  LIN {X 2625.059,Y -2566.499,Z 65.775,A 88.24449,B 0.00000,C 180.00000} ; preinsert
  LIN {X 2625.059,Y -2566.499,Z -184.225,A 88.24449,B 0.00000,C 180.00000} ; insert
  LIN {X 2625.059,Y -2566.499,Z -184.225,A 88.24449,B 0.00000,C 180.00000} ; release
  LIN {X 2625.059,Y -2566.499,Z 115.775,A 88.24449,B 0.00000,C 180.00000} ; retreat
  ; Step 1793, bar 2402
  LIN {X 1875.059,Y -2566.499,Z 1020.471,A 88.24449,B 0.00000,C 180.00000} ; outside
  LIN {X 1875.059,Y -2566.499,Z 65.775,A 88.24449,B 0.00000,C 180.00000} ; preinsert
  LIN {X 1875.059,Y -2566.499,Z -184.225,A 88.24449,B 0.00000,C 180.00000} ; insert
  LIN {X 1875.059,Y -2566.499,Z -184.225,A 88.24449,B 0.00000,C 180.00000} ; release
  LIN {X 1875.059,Y -2566.499,Z 115.775,A 88.24449,B 0.00000,C 180.00000} ; retreat
  ; Step 1794, bar 2396
  LIN {X 1125.059,Y -2566.499,Z 1020.471,A 88.24449,B 0.00000,C 180.00000} ; outside
  LIN {X 1125.059,Y -2566.499,Z 65.775,A 88.24449,B 0.00000,C 180.00000} ; preinsert
  LIN {X 1125.059,Y -2566.499,Z -184.225,A 88.24449,B 0.00000,C 180.00000} ; insert
  LIN {X 1125.059,Y -2566.499,Z -184.225,A 88.24449,B 0.00000,C 180.00000} ; release
  LIN {X 1125.059,Y -2566.499,Z 115.775,A 88.24449,B 0.00000,C 180.00000} ; retreat
  ; Step 1795, bar 2391
  LIN {X 375.059,Y -2566.499,Z 1020.471,A 88.24449,B 0.00000,C 180.00000} ; outside
  LIN {X 375.059,Y -2566.499,Z 65.775,A 88.24449,B 0.00000,C 180.00000} ; preinsert
  LIN {X 375.059,Y -2566.499,Z -184.225,A 88.24449,B 0.00000,C 180.00000} ; insert
  LIN {X 375.059,Y -2566.499,Z -184.225,A 88.24449,B 0.00000,C 180.00000} ; release
  LIN {X 375.059,Y -2566.499,Z 115.775,A 88.24449,B 0.00000,C 180.00000} ; retreat
  ; Step 1796, bar 2106
  LIN {X -15850.059,Y 2566.499,Z 1020.471,A -91.75551,B 0.00000,C -180.00000} ; outside
  LIN {X -15850.059,Y 2566.499,Z 65.775,A -91.75551,B 0.00000,C -180.00000} ; preinsert
  LIN {X -15850.059,Y 2566.499,Z -184.225,A -91.75551,B 0.00000,C -180.00000} ; insert
  LIN {X -15850.059,Y 2566.499,Z -184.225,A -91.75551,B 0.00000,C -180.00000} ; release
  LIN {X -15850.059,Y 2566.499,Z 115.775,A -91.75551,B 0.00000,C -180.00000} ; retreat
  ; Step 1797, bar 2100
  LIN {X -15250.059,Y 2566.499,Z 1020.471,A -91.75551,B 0.00000,C -180.00000} ; outside
  LIN {X -15250.059,Y 2566.499,Z 65.775,A -91.75551,B 0.00000,C -180.00000} ; preinsert
  LIN {X -15250.059,Y 2566.499,Z -184.225,A -91.75551,B 0.00000,C -180.00000} ; insert
  LIN {X -15250.059,Y 2566.499,Z -184.225,A -91.75551,B 0.00000,C -180.00000} ; release
  LIN {X -15250.059,Y 2566.499,Z 115.775,A -91.75551,B 0.00000,C -180.00000} ; retreat
  ; Step 1798, bar 2094
  LIN {X -14650.059,Y 2566.499,Z 1020.471,A -91.75551,B 0.00000,C -180.00000} ; outside
  LIN {X -14650.059,Y 2566.499,Z 65.775,A -91.75551,B 0.00000,C -180.00000} ; preinsert
  LIN {X -14650.059,Y 2566.499,Z -184.225,A -91.75551,B 0.00000,C -180.00000} ; insert
  LIN {X -14650.059,Y 2566.499,Z -184.225,A -91.75551,B 0.00000,C -180.00000} ; release
  LIN {X -14650.059,Y 2566.499,Z 115.775,A -91.75551,B 0.00000,C -180.00000} ; retreat
  ; Step 1799, bar 2088
  LIN {X -14050.059,Y 2566.499,Z 1020.471,A -91.75551,B 0.00000,C -180.00000} ; outside
  LIN {X -14050.059,Y 2566.499,Z 65.775,A -91.75551,B 0.00000,C -180.00000} ; preinsert
  LIN {X -14050.059,Y 2566.499,Z -184.225,A -91.75551,B 0.00000,C -180.00000} ; insert
  LIN {X -14050.059,Y 2566.499,Z -184.225,A -91.75551,B 0.00000,C -180.00000} ; release
  LIN {X -14050.059,Y 2566.499,Z 115.775,A -91.75551,B 0.00000,C -180.00000} ; retreat
  ; Step 1800, bar 2082
  LIN {X -13450.059,Y 2566.499,Z 1020.471,A -91.75551,B 0.00000,C -180.00000} ; outside
  LIN {X -13450.059,Y 2566.499,Z 65.775,A -91.75551,B 0.00000,C -180.00000} ; preinsert
  LIN {X -13450.059,Y 2566.499,Z -184.225,A -91.75551,B 0.00000,C -180.00000} ; insert
  LIN {X -13450.059,Y 2566.499,Z -184.225,A -91.75551,B 0.00000,C -180.00000} ; release
  LIN {X -13450.059,Y 2566.499,Z 115.775,A -91.75551,B 0.00000,C -180.00000} ; retreat
  ; Step 1801, bar 2076
  LIN {X -12850.059,Y 2566.499,Z 1020.471,A -91.75551,B 0.00000,C -180.00000} ; outside
  LIN {X -12850.059,Y 2566.499,Z 65.775,A -91.75551,B 0.00000,C -180.00000} ; preinsert
  LIN {X -12850.059,Y 2566.499,Z -184.225,A -91.75551,B 0.00000,C -180.00000} ; insert
  LIN {X -12850.059,Y 2566.499,Z -184.225,A -91.75551,B 0.00000,C -180.00000} ; release
  LIN {X -12850.059,Y 2566.499,Z 115.775,A -91.75551,B 0.00000,C -180.00000} ; retreat
  ; Step 1802, bar 2069
  LIN {X -12250.059,Y 2566.499,Z 1020.471,A -91.75551,B 0.00000,C -180.00000} ; outside
  LIN {X -12250.059,Y 2566.499,Z 65.775,A -91.75551,B 0.00000,C -180.00000} ; preinsert
  LIN {X -12250.059,Y 2566.499,Z -184.225,A -91.75551,B 0.00000,C -180.00000} ; insert
  LIN {X -12250.059,Y 2566.499,Z -184.225,A -91.75551,B 0.00000,C -180.00000} ; release
  LIN {X -12250.059,Y 2566.499,Z 115.775,A -91.75551,B 0.00000,C -180.00000} ; retreat
  ; Step 1803, bar 2063
  LIN {X -11625.059,Y 2566.499,Z 1020.471,A -91.75551,B 0.00000,C -180.00000} ; outside
  LIN {X -11625.059,Y 2566.499,Z 65.775,A -91.75551,B 0.00000,C -180.00000} ; preinsert
  LIN {X -11625.059,Y 2566.499,Z -184.225,A -91.75551,B 0.00000,C -180.00000} ; insert
  LIN {X -11625.059,Y 2566.499,Z -184.225,A -91.75551,B 0.00000,C -180.00000} ; release
  LIN {X -11625.059,Y 2566.499,Z 115.775,A -91.75551,B 0.00000,C -180.00000} ; retreat
  ; Step 1804, bar 2057
  LIN {X -10875.059,Y 2566.499,Z 1020.471,A -91.75551,B 0.00000,C -180.00000} ; outside
  LIN {X -10875.059,Y 2566.499,Z 65.775,A -91.75551,B 0.00000,C -180.00000} ; preinsert
  LIN {X -10875.059,Y 2566.499,Z -184.225,A -91.75551,B 0.00000,C -180.00000} ; insert
  LIN {X -10875.059,Y 2566.499,Z -184.225,A -91.75551,B 0.00000,C -180.00000} ; release
  LIN {X -10875.059,Y 2566.499,Z 115.775,A -91.75551,B 0.00000,C -180.00000} ; retreat
  ; Step 1805, bar 2051
  LIN {X -10125.059,Y 2566.499,Z 1020.471,A -91.75551,B 0.00000,C -180.00000} ; outside
  LIN {X -10125.059,Y 2566.499,Z 65.775,A -91.75551,B 0.00000,C -180.00000} ; preinsert
  LIN {X -10125.059,Y 2566.499,Z -184.225,A -91.75551,B 0.00000,C -180.00000} ; insert
  LIN {X -10125.059,Y 2566.499,Z -184.225,A -91.75551,B 0.00000,C -180.00000} ; release
  LIN {X -10125.059,Y 2566.499,Z 115.775,A -91.75551,B 0.00000,C -180.00000} ; retreat
  ; Step 1806, bar 2045
  LIN {X -9375.059,Y 2566.499,Z 1020.471,A -91.75551,B 0.00000,C -180.00000} ; outside
  LIN {X -9375.059,Y 2566.499,Z 65.775,A -91.75551,B 0.00000,C -180.00000} ; preinsert
  LIN {X -9375.059,Y 2566.499,Z -184.225,A -91.75551,B 0.00000,C -180.00000} ; insert
  LIN {X -9375.059,Y 2566.499,Z -184.225,A -91.75551,B 0.00000,C -180.00000} ; release
  LIN {X -9375.059,Y 2566.499,Z 115.775,A -91.75551,B 0.00000,C -180.00000} ; retreat
  ; Step 1807, bar 2039
  LIN {X -8625.059,Y 2566.499,Z 1020.471,A -91.75551,B 0.00000,C -180.00000} ; outside
  LIN {X -8625.059,Y 2566.499,Z 65.775,A -91.75551,B 0.00000,C -180.00000} ; preinsert
  LIN {X -8625.059,Y 2566.499,Z -184.225,A -91.75551,B 0.00000,C -180.00000} ; insert
  LIN {X -8625.059,Y 2566.499,Z -184.225,A -91.75551,B 0.00000,C -180.00000} ; release
  LIN {X -8625.059,Y 2566.499,Z 115.775,A -91.75551,B 0.00000,C -180.00000} ; retreat
  ; Step 1808, bar 2033
  LIN {X -7875.059,Y 2566.499,Z 1020.471,A -91.75551,B 0.00000,C -180.00000} ; outside
  LIN {X -7875.059,Y 2566.499,Z 65.775,A -91.75551,B 0.00000,C -180.00000} ; preinsert
  LIN {X -7875.059,Y 2566.499,Z -184.225,A -91.75551,B 0.00000,C -180.00000} ; insert
  LIN {X -7875.059,Y 2566.499,Z -184.225,A -91.75551,B 0.00000,C -180.00000} ; release
  LIN {X -7875.059,Y 2566.499,Z 115.775,A -91.75551,B 0.00000,C -180.00000} ; retreat
  ; Step 1809, bar 2027
  LIN {X -7125.059,Y 2566.499,Z 1020.471,A -91.75551,B 0.00000,C -180.00000} ; outside
  LIN {X -7125.059,Y 2566.499,Z 65.775,A -91.75551,B 0.00000,C -180.00000} ; preinsert
  LIN {X -7125.059,Y 2566.499,Z -184.225,A -91.75551,B 0.00000,C -180.00000} ; insert
  LIN {X -7125.059,Y 2566.499,Z -184.225,A -91.75551,B 0.00000,C -180.00000} ; release
  LIN {X -7125.059,Y 2566.499,Z 115.775,A -91.75551,B 0.00000,C -180.00000} ; retreat
  ; Step 1810, bar 2021
  LIN {X -6375.059,Y 2566.499,Z 1020.471,A -91.75551,B 0.00000,C -180.00000} ; outside
  LIN {X -6375.059,Y 2566.499,Z 65.775,A -91.75551,B 0.00000,C -180.00000} ; preinsert
  LIN {X -6375.059,Y 2566.499,Z -184.225,A -91.75551,B 0.00000,C -180.00000} ; insert
  LIN {X -6375.059,Y 2566.499,Z -184.225,A -91.75551,B 0.00000,C -180.00000} ; release
  LIN {X -6375.059,Y 2566.499,Z 115.775,A -91.75551,B 0.00000,C -180.00000} ; retreat
  ; Step 1811, bar 2015
  LIN {X -5625.059,Y 2566.499,Z 1020.471,A -91.75551,B 0.00000,C -180.00000} ; outside
  LIN {X -5625.059,Y 2566.499,Z 65.775,A -91.75551,B 0.00000,C -180.00000} ; preinsert
  LIN {X -5625.059,Y 2566.499,Z -184.225,A -91.75551,B 0.00000,C -180.00000} ; insert
  LIN {X -5625.059,Y 2566.499,Z -184.225,A -91.75551,B 0.00000,C -180.00000} ; release
  LIN {X -5625.059,Y 2566.499,Z 115.775,A -91.75551,B 0.00000,C -180.00000} ; retreat
  ; Step 1812, bar 2009
  LIN {X -4875.059,Y 2566.499,Z 1020.471,A -91.75551,B 0.00000,C -180.00000} ; outside
  LIN {X -4875.059,Y 2566.499,Z 65.775,A -91.75551,B 0.00000,C -180.00000} ; preinsert
  LIN {X -4875.059,Y 2566.499,Z -184.225,A -91.75551,B 0.00000,C -180.00000} ; insert
  LIN {X -4875.059,Y 2566.499,Z -184.225,A -91.75551,B 0.00000,C -180.00000} ; release
  LIN {X -4875.059,Y 2566.499,Z 115.775,A -91.75551,B 0.00000,C -180.00000} ; retreat
  ; Step 1813, bar 2003
  LIN {X -4125.059,Y 2566.499,Z 1020.471,A -91.75551,B 0.00000,C -180.00000} ; outside
  LIN {X -4125.059,Y 2566.499,Z 65.775,A -91.75551,B 0.00000,C -180.00000} ; preinsert
  LIN {X -4125.059,Y 2566.499,Z -184.225,A -91.75551,B 0.00000,C -180.00000} ; insert
  LIN {X -4125.059,Y 2566.499,Z -184.225,A -91.75551,B 0.00000,C -180.00000} ; release
  LIN {X -4125.059,Y 2566.499,Z 115.775,A -91.75551,B 0.00000,C -180.00000} ; retreat
  ; Step 1814, bar 1997
  LIN {X -3375.059,Y 2566.499,Z 1020.471,A -91.75551,B 0.00000,C -180.00000} ; outside
  LIN {X -3375.059,Y 2566.499,Z 65.775,A -91.75551,B 0.00000,C -180.00000} ; preinsert
  LIN {X -3375.059,Y 2566.499,Z -184.225,A -91.75551,B 0.00000,C -180.00000} ; insert
  LIN {X -3375.059,Y 2566.499,Z -184.225,A -91.75551,B 0.00000,C -180.00000} ; release
  LIN {X -3375.059,Y 2566.499,Z 115.775,A -91.75551,B 0.00000,C -180.00000} ; retreat
  ; Step 1815, bar 1991
  LIN {X -2625.059,Y 2566.499,Z 1020.471,A -91.75551,B 0.00000,C -180.00000} ; outside
  LIN {X -2625.059,Y 2566.499,Z 65.775,A -91.75551,B 0.00000,C -180.00000} ; preinsert
  LIN {X -2625.059,Y 2566.499,Z -184.225,A -91.75551,B 0.00000,C -180.00000} ; insert
  LIN {X -2625.059,Y 2566.499,Z -184.225,A -91.75551,B 0.00000,C -180.00000} ; release
  LIN {X -2625.059,Y 2566.499,Z 115.775,A -91.75551,B 0.00000,C -180.00000} ; retreat
  ; Step 1816, bar 1985
  LIN {X -1875.059,Y 2566.499,Z 1020.471,A -91.75551,B 0.00000,C -180.00000} ; outside
  LIN {X -1875.059,Y 2566.499,Z 65.775,A -91.75551,B 0.00000,C -180.00000} ; preinsert
  LIN {X -1875.059,Y 2566.499,Z -184.225,A -91.75551,B 0.00000,C -180.00000} ; insert
  LIN {X -1875.059,Y 2566.499,Z -184.225,A -91.75551,B 0.00000,C -180.00000} ; release
  LIN {X -1875.059,Y 2566.499,Z 115.775,A -91.75551,B 0.00000,C -180.00000} ; retreat
  ; Step 1817, bar 1979
  LIN {X -1125.059,Y 2566.499,Z 1020.471,A -91.75551,B 0.00000,C -180.00000} ; outside
  LIN {X -1125.059,Y 2566.499,Z 65.775,A -91.75551,B 0.00000,C -180.00000} ; preinsert
  LIN {X -1125.059,Y 2566.499,Z -184.225,A -91.75551,B 0.00000,C -180.00000} ; insert
  LIN {X -1125.059,Y 2566.499,Z -184.225,A -91.75551,B 0.00000,C -180.00000} ; release
  LIN {X -1125.059,Y 2566.499,Z 115.775,A -91.75551,B 0.00000,C -180.00000} ; retreat
  ; Step 1818, bar 1966
  LIN {X -375.059,Y 2566.499,Z 1020.471,A -91.75551,B 0.00000,C -180.00000} ; outside
  LIN {X -375.059,Y 2566.499,Z 65.775,A -91.75551,B 0.00000,C -180.00000} ; preinsert
  LIN {X -375.059,Y 2566.499,Z -184.225,A -91.75551,B 0.00000,C -180.00000} ; insert
  LIN {X -375.059,Y 2566.499,Z -184.225,A -91.75551,B 0.00000,C -180.00000} ; release
  LIN {X -375.059,Y 2566.499,Z 115.775,A -91.75551,B 0.00000,C -180.00000} ; retreat
  ; Step 1819, bar 882
  LIN {X -16231.996,Y -2667.355,Z 1143.930,A -89.99946,B 0.00000,C 180.00000} ; outside
  LIN {X -16231.996,Y -2667.355,Z 190.712,A -89.99946,B 0.00000,C 180.00000} ; preinsert
  LIN {X -16231.996,Y -2667.355,Z -59.288,A -89.99946,B 0.00000,C 180.00000} ; insert
  LIN {X -16231.996,Y -2667.355,Z -59.288,A -89.99946,B 0.00000,C 180.00000} ; release
  LIN {X -16231.996,Y -2667.355,Z 240.712,A -89.99946,B 0.00000,C 180.00000} ; retreat
  ; Step 1820, bar 880
  LIN {X -16131.996,Y -2667.355,Z 1143.930,A -89.99946,B 0.00000,C 180.00000} ; outside
  LIN {X -16131.996,Y -2667.355,Z 190.712,A -89.99946,B 0.00000,C 180.00000} ; preinsert
  LIN {X -16131.996,Y -2667.355,Z -59.288,A -89.99946,B 0.00000,C 180.00000} ; insert
  LIN {X -16131.996,Y -2667.355,Z -59.288,A -89.99946,B 0.00000,C 180.00000} ; release
  LIN {X -16131.996,Y -2667.355,Z 240.712,A -89.99946,B 0.00000,C 180.00000} ; retreat
  ; Step 1821, bar 878
  LIN {X -16031.996,Y -2667.355,Z 1143.930,A -89.99946,B 0.00000,C 180.00000} ; outside
  LIN {X -16031.996,Y -2667.355,Z 190.712,A -89.99946,B 0.00000,C 180.00000} ; preinsert
  LIN {X -16031.996,Y -2667.355,Z -59.288,A -89.99946,B 0.00000,C 180.00000} ; insert
  LIN {X -16031.996,Y -2667.355,Z -59.288,A -89.99946,B 0.00000,C 180.00000} ; release
  LIN {X -16031.996,Y -2667.355,Z 240.712,A -89.99946,B 0.00000,C 180.00000} ; retreat
  ; Step 1822, bar 876
  LIN {X -15931.996,Y -2667.355,Z 1143.930,A -89.99946,B 0.00000,C 180.00000} ; outside
  LIN {X -15931.996,Y -2667.355,Z 190.712,A -89.99946,B 0.00000,C 180.00000} ; preinsert
  LIN {X -15931.996,Y -2667.355,Z -59.288,A -89.99946,B 0.00000,C 180.00000} ; insert
  LIN {X -15931.996,Y -2667.355,Z -59.288,A -89.99946,B 0.00000,C 180.00000} ; release
  LIN {X -15931.996,Y -2667.355,Z 240.712,A -89.99946,B 0.00000,C 180.00000} ; retreat
  ; Step 1823, bar 874
  LIN {X -15831.996,Y -2667.355,Z 1143.930,A -89.99946,B 0.00000,C 180.00000} ; outside
  LIN {X -15831.996,Y -2667.355,Z 190.712,A -89.99946,B 0.00000,C 180.00000} ; preinsert
  LIN {X -15831.996,Y -2667.355,Z -59.288,A -89.99946,B 0.00000,C 180.00000} ; insert
  LIN {X -15831.996,Y -2667.355,Z -59.288,A -89.99946,B 0.00000,C 180.00000} ; release
  LIN {X -15831.996,Y -2667.355,Z 240.712,A -89.99946,B 0.00000,C 180.00000} ; retreat
  ; Step 1824, bar 872
  LIN {X -15731.996,Y -2667.355,Z 1143.930,A -89.99946,B 0.00000,C 180.00000} ; outside
  LIN {X -15731.996,Y -2667.355,Z 190.712,A -89.99946,B 0.00000,C 180.00000} ; preinsert
  LIN {X -15731.996,Y -2667.355,Z -59.288,A -89.99946,B 0.00000,C 180.00000} ; insert
  LIN {X -15731.996,Y -2667.355,Z -59.288,A -89.99946,B 0.00000,C 180.00000} ; release
  LIN {X -15731.996,Y -2667.355,Z 240.712,A -89.99946,B 0.00000,C 180.00000} ; retreat
  ; Step 1825, bar 870
  LIN {X -15631.996,Y -2667.355,Z 1143.930,A -89.99946,B 0.00000,C 180.00000} ; outside
  LIN {X -15631.996,Y -2667.355,Z 190.712,A -89.99946,B 0.00000,C 180.00000} ; preinsert
  LIN {X -15631.996,Y -2667.355,Z -59.288,A -89.99946,B 0.00000,C 180.00000} ; insert
  LIN {X -15631.996,Y -2667.355,Z -59.288,A -89.99946,B 0.00000,C 180.00000} ; release
  LIN {X -15631.996,Y -2667.355,Z 240.712,A -89.99946,B 0.00000,C 180.00000} ; retreat
  ; Step 1826, bar 868
  LIN {X -15531.996,Y -2667.355,Z 1143.930,A -89.99946,B 0.00000,C 180.00000} ; outside
  LIN {X -15531.996,Y -2667.355,Z 190.712,A -89.99946,B 0.00000,C 180.00000} ; preinsert
  LIN {X -15531.996,Y -2667.355,Z -59.288,A -89.99946,B 0.00000,C 180.00000} ; insert
  LIN {X -15531.996,Y -2667.355,Z -59.288,A -89.99946,B 0.00000,C 180.00000} ; release
  LIN {X -15531.996,Y -2667.355,Z 240.712,A -89.99946,B 0.00000,C 180.00000} ; retreat
  ; Step 1827, bar 866
  LIN {X -15431.996,Y -2667.355,Z 1143.930,A -89.99946,B 0.00000,C 180.00000} ; outside
  LIN {X -15431.996,Y -2667.355,Z 190.712,A -89.99946,B 0.00000,C 180.00000} ; preinsert
  LIN {X -15431.996,Y -2667.355,Z -59.288,A -89.99946,B 0.00000,C 180.00000} ; insert
  LIN {X -15431.996,Y -2667.355,Z -59.288,A -89.99946,B 0.00000,C 180.00000} ; release
  LIN {X -15431.996,Y -2667.355,Z 240.712,A -89.99946,B 0.00000,C 180.00000} ; retreat
  ; Step 1828, bar 864
  LIN {X -15331.996,Y -2667.355,Z 1143.930,A -89.99946,B 0.00000,C 180.00000} ; outside
  LIN {X -15331.996,Y -2667.355,Z 190.712,A -89.99946,B 0.00000,C 180.00000} ; preinsert
  LIN {X -15331.996,Y -2667.355,Z -59.288,A -89.99946,B 0.00000,C 180.00000} ; insert
  LIN {X -15331.996,Y -2667.355,Z -59.288,A -89.99946,B 0.00000,C 180.00000} ; release
  LIN {X -15331.996,Y -2667.355,Z 240.712,A -89.99946,B 0.00000,C 180.00000} ; retreat
  ; Step 1829, bar 862
  LIN {X -15231.996,Y -2667.355,Z 1143.930,A -89.99946,B 0.00000,C 180.00000} ; outside
  LIN {X -15231.996,Y -2667.355,Z 190.712,A -89.99946,B 0.00000,C 180.00000} ; preinsert
  LIN {X -15231.996,Y -2667.355,Z -59.288,A -89.99946,B 0.00000,C 180.00000} ; insert
  LIN {X -15231.996,Y -2667.355,Z -59.288,A -89.99946,B 0.00000,C 180.00000} ; release
  LIN {X -15231.996,Y -2667.355,Z 240.712,A -89.99946,B 0.00000,C 180.00000} ; retreat
  ; Step 1830, bar 860
  LIN {X -15131.996,Y -2667.355,Z 1143.930,A -89.99946,B 0.00000,C 180.00000} ; outside
  LIN {X -15131.996,Y -2667.355,Z 190.712,A -89.99946,B 0.00000,C 180.00000} ; preinsert
  LIN {X -15131.996,Y -2667.355,Z -59.288,A -89.99946,B 0.00000,C 180.00000} ; insert
  LIN {X -15131.996,Y -2667.355,Z -59.288,A -89.99946,B 0.00000,C 180.00000} ; release
  LIN {X -15131.996,Y -2667.355,Z 240.712,A -89.99946,B 0.00000,C 180.00000} ; retreat
  ; Step 1831, bar 858
  LIN {X -15031.996,Y -2667.355,Z 1143.930,A -89.99946,B 0.00000,C 180.00000} ; outside
  LIN {X -15031.996,Y -2667.355,Z 190.712,A -89.99946,B 0.00000,C 180.00000} ; preinsert
  LIN {X -15031.996,Y -2667.355,Z -59.288,A -89.99946,B 0.00000,C 180.00000} ; insert
  LIN {X -15031.996,Y -2667.355,Z -59.288,A -89.99946,B 0.00000,C 180.00000} ; release
  LIN {X -15031.996,Y -2667.355,Z 240.712,A -89.99946,B 0.00000,C 180.00000} ; retreat
  ; Step 1832, bar 856
  LIN {X -14931.996,Y -2667.355,Z 1143.930,A -89.99946,B 0.00000,C 180.00000} ; outside
  LIN {X -14931.996,Y -2667.355,Z 190.712,A -89.99946,B 0.00000,C 180.00000} ; preinsert
  LIN {X -14931.996,Y -2667.355,Z -59.288,A -89.99946,B 0.00000,C 180.00000} ; insert
  LIN {X -14931.996,Y -2667.355,Z -59.288,A -89.99946,B 0.00000,C 180.00000} ; release
  LIN {X -14931.996,Y -2667.355,Z 240.712,A -89.99946,B 0.00000,C 180.00000} ; retreat
  ; Step 1833, bar 854
  LIN {X -14831.996,Y -2667.355,Z 1143.930,A -89.99946,B 0.00000,C 180.00000} ; outside
  LIN {X -14831.996,Y -2667.355,Z 190.712,A -89.99946,B 0.00000,C 180.00000} ; preinsert
  LIN {X -14831.996,Y -2667.355,Z -59.288,A -89.99946,B 0.00000,C 180.00000} ; insert
  LIN {X -14831.996,Y -2667.355,Z -59.288,A -89.99946,B 0.00000,C 180.00000} ; release
  LIN {X -14831.996,Y -2667.355,Z 240.712,A -89.99946,B 0.00000,C 180.00000} ; retreat
  ; Step 1834, bar 852
  LIN {X -14731.996,Y -2667.355,Z 1143.930,A -89.99946,B 0.00000,C 180.00000} ; outside
  LIN {X -14731.996,Y -2667.355,Z 190.712,A -89.99946,B 0.00000,C 180.00000} ; preinsert
  LIN {X -14731.996,Y -2667.355,Z -59.288,A -89.99946,B 0.00000,C 180.00000} ; insert
  LIN {X -14731.996,Y -2667.355,Z -59.288,A -89.99946,B 0.00000,C 180.00000} ; release
  LIN {X -14731.996,Y -2667.355,Z 240.712,A -89.99946,B 0.00000,C 180.00000} ; retreat
  ; Step 1835, bar 850
  LIN {X -14631.996,Y -2667.355,Z 1143.930,A -89.99946,B 0.00000,C 180.00000} ; outside
  LIN {X -14631.996,Y -2667.355,Z 190.712,A -89.99946,B 0.00000,C 180.00000} ; preinsert
  LIN {X -14631.996,Y -2667.355,Z -59.288,A -89.99946,B 0.00000,C 180.00000} ; insert
  LIN {X -14631.996,Y -2667.355,Z -59.288,A -89.99946,B 0.00000,C 180.00000} ; release
  LIN {X -14631.996,Y -2667.355,Z 240.712,A -89.99946,B 0.00000,C 180.00000} ; retreat
  ; Step 1836, bar 848
  LIN {X -14531.996,Y -2667.355,Z 1143.930,A -89.99946,B 0.00000,C 180.00000} ; outside
  LIN {X -14531.996,Y -2667.355,Z 190.712,A -89.99946,B 0.00000,C 180.00000} ; preinsert
  LIN {X -14531.996,Y -2667.355,Z -59.288,A -89.99946,B 0.00000,C 180.00000} ; insert
  LIN {X -14531.996,Y -2667.355,Z -59.288,A -89.99946,B 0.00000,C 180.00000} ; release
  LIN {X -14531.996,Y -2667.355,Z 240.712,A -89.99946,B 0.00000,C 180.00000} ; retreat
  ; Step 1837, bar 846
  LIN {X -14431.996,Y -2667.355,Z 1143.930,A -89.99946,B 0.00000,C 180.00000} ; outside
  LIN {X -14431.996,Y -2667.355,Z 190.712,A -89.99946,B 0.00000,C 180.00000} ; preinsert
  LIN {X -14431.996,Y -2667.355,Z -59.288,A -89.99946,B 0.00000,C 180.00000} ; insert
  LIN {X -14431.996,Y -2667.355,Z -59.288,A -89.99946,B 0.00000,C 180.00000} ; release
  LIN {X -14431.996,Y -2667.355,Z 240.712,A -89.99946,B 0.00000,C 180.00000} ; retreat
  ; Step 1838, bar 844
  LIN {X -14331.996,Y -2667.355,Z 1143.930,A -89.99946,B 0.00000,C 180.00000} ; outside
  LIN {X -14331.996,Y -2667.355,Z 190.712,A -89.99946,B 0.00000,C 180.00000} ; preinsert
  LIN {X -14331.996,Y -2667.355,Z -59.288,A -89.99946,B 0.00000,C 180.00000} ; insert
  LIN {X -14331.996,Y -2667.355,Z -59.288,A -89.99946,B 0.00000,C 180.00000} ; release
  LIN {X -14331.996,Y -2667.355,Z 240.712,A -89.99946,B 0.00000,C 180.00000} ; retreat
  ; Step 1839, bar 842
  LIN {X -14231.996,Y -2667.355,Z 1143.930,A -89.99946,B 0.00000,C 180.00000} ; outside
  LIN {X -14231.996,Y -2667.355,Z 190.712,A -89.99946,B 0.00000,C 180.00000} ; preinsert
  LIN {X -14231.996,Y -2667.355,Z -59.288,A -89.99946,B 0.00000,C 180.00000} ; insert
  LIN {X -14231.996,Y -2667.355,Z -59.288,A -89.99946,B 0.00000,C 180.00000} ; release
  LIN {X -14231.996,Y -2667.355,Z 240.712,A -89.99946,B 0.00000,C 180.00000} ; retreat
  ; Step 1840, bar 840
  LIN {X -14131.996,Y -2667.355,Z 1143.930,A -89.99946,B 0.00000,C 180.00000} ; outside
  LIN {X -14131.996,Y -2667.355,Z 190.712,A -89.99946,B 0.00000,C 180.00000} ; preinsert
  LIN {X -14131.996,Y -2667.355,Z -59.288,A -89.99946,B 0.00000,C 180.00000} ; insert
  LIN {X -14131.996,Y -2667.355,Z -59.288,A -89.99946,B 0.00000,C 180.00000} ; release
  LIN {X -14131.996,Y -2667.355,Z 240.712,A -89.99946,B 0.00000,C 180.00000} ; retreat
  ; Step 1841, bar 838
  LIN {X -13831.996,Y -2667.355,Z 1143.930,A -89.99946,B 0.00000,C 180.00000} ; outside
  LIN {X -13831.996,Y -2667.355,Z 190.712,A -89.99946,B 0.00000,C 180.00000} ; preinsert
  LIN {X -13831.996,Y -2667.355,Z -59.288,A -89.99946,B 0.00000,C 180.00000} ; insert
  LIN {X -13831.996,Y -2667.355,Z -59.288,A -89.99946,B 0.00000,C 180.00000} ; release
  LIN {X -13831.996,Y -2667.355,Z 240.712,A -89.99946,B 0.00000,C 180.00000} ; retreat
  ; Step 1842, bar 836
  LIN {X -13731.996,Y -2667.355,Z 1143.930,A -89.99946,B 0.00000,C 180.00000} ; outside
  LIN {X -13731.996,Y -2667.355,Z 190.712,A -89.99946,B 0.00000,C 180.00000} ; preinsert
  LIN {X -13731.996,Y -2667.355,Z -59.288,A -89.99946,B 0.00000,C 180.00000} ; insert
  LIN {X -13731.996,Y -2667.355,Z -59.288,A -89.99946,B 0.00000,C 180.00000} ; release
  LIN {X -13731.996,Y -2667.355,Z 240.712,A -89.99946,B 0.00000,C 180.00000} ; retreat
  ; Step 1843, bar 834
  LIN {X -13631.996,Y -2667.355,Z 1143.930,A -89.99946,B 0.00000,C 180.00000} ; outside
  LIN {X -13631.996,Y -2667.355,Z 190.712,A -89.99946,B 0.00000,C 180.00000} ; preinsert
  LIN {X -13631.996,Y -2667.355,Z -59.288,A -89.99946,B 0.00000,C 180.00000} ; insert
  LIN {X -13631.996,Y -2667.355,Z -59.288,A -89.99946,B 0.00000,C 180.00000} ; release
  LIN {X -13631.996,Y -2667.355,Z 240.712,A -89.99946,B 0.00000,C 180.00000} ; retreat
  ; Step 1844, bar 832
  LIN {X -13531.996,Y -2667.355,Z 1143.930,A -89.99946,B 0.00000,C 180.00000} ; outside
  LIN {X -13531.996,Y -2667.355,Z 190.712,A -89.99946,B 0.00000,C 180.00000} ; preinsert
  LIN {X -13531.996,Y -2667.355,Z -59.288,A -89.99946,B 0.00000,C 180.00000} ; insert
  LIN {X -13531.996,Y -2667.355,Z -59.288,A -89.99946,B 0.00000,C 180.00000} ; release
  LIN {X -13531.996,Y -2667.355,Z 240.712,A -89.99946,B 0.00000,C 180.00000} ; retreat
  ; Step 1845, bar 830
  LIN {X -13431.996,Y -2667.355,Z 1143.930,A -89.99946,B 0.00000,C 180.00000} ; outside
  LIN {X -13431.996,Y -2667.355,Z 190.712,A -89.99946,B 0.00000,C 180.00000} ; preinsert
  LIN {X -13431.996,Y -2667.355,Z -59.288,A -89.99946,B 0.00000,C 180.00000} ; insert
  LIN {X -13431.996,Y -2667.355,Z -59.288,A -89.99946,B 0.00000,C 180.00000} ; release
  LIN {X -13431.996,Y -2667.355,Z 240.712,A -89.99946,B 0.00000,C 180.00000} ; retreat
  ; Step 1846, bar 828
  LIN {X -13331.996,Y -2667.355,Z 1143.930,A -89.99946,B 0.00000,C 180.00000} ; outside
  LIN {X -13331.996,Y -2667.355,Z 190.712,A -89.99946,B 0.00000,C 180.00000} ; preinsert
  LIN {X -13331.996,Y -2667.355,Z -59.288,A -89.99946,B 0.00000,C 180.00000} ; insert
  LIN {X -13331.996,Y -2667.355,Z -59.288,A -89.99946,B 0.00000,C 180.00000} ; release
  LIN {X -13331.996,Y -2667.355,Z 240.712,A -89.99946,B 0.00000,C 180.00000} ; retreat
  ; Step 1847, bar 826
  LIN {X -13231.996,Y -2667.355,Z 1143.930,A -89.99946,B 0.00000,C 180.00000} ; outside
  LIN {X -13231.996,Y -2667.355,Z 190.712,A -89.99946,B 0.00000,C 180.00000} ; preinsert
  LIN {X -13231.996,Y -2667.355,Z -59.288,A -89.99946,B 0.00000,C 180.00000} ; insert
  LIN {X -13231.996,Y -2667.355,Z -59.288,A -89.99946,B 0.00000,C 180.00000} ; release
  LIN {X -13231.996,Y -2667.355,Z 240.712,A -89.99946,B 0.00000,C 180.00000} ; retreat
  ; Step 1848, bar 824
  LIN {X -13131.996,Y -2667.355,Z 1143.930,A -89.99946,B 0.00000,C 180.00000} ; outside
  LIN {X -13131.996,Y -2667.355,Z 190.712,A -89.99946,B 0.00000,C 180.00000} ; preinsert
  LIN {X -13131.996,Y -2667.355,Z -59.288,A -89.99946,B 0.00000,C 180.00000} ; insert
  LIN {X -13131.996,Y -2667.355,Z -59.288,A -89.99946,B 0.00000,C 180.00000} ; release
  LIN {X -13131.996,Y -2667.355,Z 240.712,A -89.99946,B 0.00000,C 180.00000} ; retreat
  ; Step 1849, bar 822
  LIN {X -13031.996,Y -2667.355,Z 1143.930,A -89.99946,B 0.00000,C 180.00000} ; outside
  LIN {X -13031.996,Y -2667.355,Z 190.712,A -89.99946,B 0.00000,C 180.00000} ; preinsert
  LIN {X -13031.996,Y -2667.355,Z -59.288,A -89.99946,B 0.00000,C 180.00000} ; insert
  LIN {X -13031.996,Y -2667.355,Z -59.288,A -89.99946,B 0.00000,C 180.00000} ; release
  LIN {X -13031.996,Y -2667.355,Z 240.712,A -89.99946,B 0.00000,C 180.00000} ; retreat
  ; Step 1850, bar 820
  LIN {X -12931.996,Y -2667.355,Z 1143.930,A -89.99946,B 0.00000,C 180.00000} ; outside
  LIN {X -12931.996,Y -2667.355,Z 190.712,A -89.99946,B 0.00000,C 180.00000} ; preinsert
  LIN {X -12931.996,Y -2667.355,Z -59.288,A -89.99946,B 0.00000,C 180.00000} ; insert
  LIN {X -12931.996,Y -2667.355,Z -59.288,A -89.99946,B 0.00000,C 180.00000} ; release
  LIN {X -12931.996,Y -2667.355,Z 240.712,A -89.99946,B 0.00000,C 180.00000} ; retreat
  ; Step 1851, bar 818
  LIN {X -12831.996,Y -2667.355,Z 1143.930,A -89.99946,B 0.00000,C 180.00000} ; outside
  LIN {X -12831.996,Y -2667.355,Z 190.712,A -89.99946,B 0.00000,C 180.00000} ; preinsert
  LIN {X -12831.996,Y -2667.355,Z -59.288,A -89.99946,B 0.00000,C 180.00000} ; insert
  LIN {X -12831.996,Y -2667.355,Z -59.288,A -89.99946,B 0.00000,C 180.00000} ; release
  LIN {X -12831.996,Y -2667.355,Z 240.712,A -89.99946,B 0.00000,C 180.00000} ; retreat
  ; Step 1852, bar 816
  LIN {X -12731.996,Y -2667.355,Z 1143.930,A -89.99946,B 0.00000,C 180.00000} ; outside
  LIN {X -12731.996,Y -2667.355,Z 190.712,A -89.99946,B 0.00000,C 180.00000} ; preinsert
  LIN {X -12731.996,Y -2667.355,Z -59.288,A -89.99946,B 0.00000,C 180.00000} ; insert
  LIN {X -12731.996,Y -2667.355,Z -59.288,A -89.99946,B 0.00000,C 180.00000} ; release
  LIN {X -12731.996,Y -2667.355,Z 240.712,A -89.99946,B 0.00000,C 180.00000} ; retreat
  ; Step 1853, bar 814
  LIN {X -12631.996,Y -2667.355,Z 1143.930,A -89.99946,B 0.00000,C 180.00000} ; outside
  LIN {X -12631.996,Y -2667.355,Z 190.712,A -89.99946,B 0.00000,C 180.00000} ; preinsert
  LIN {X -12631.996,Y -2667.355,Z -59.288,A -89.99946,B 0.00000,C 180.00000} ; insert
  LIN {X -12631.996,Y -2667.355,Z -59.288,A -89.99946,B 0.00000,C 180.00000} ; release
  LIN {X -12631.996,Y -2667.355,Z 240.712,A -89.99946,B 0.00000,C 180.00000} ; retreat
  ; Step 1854, bar 812
  LIN {X -12531.996,Y -2667.355,Z 1143.930,A -89.99946,B 0.00000,C 180.00000} ; outside
  LIN {X -12531.996,Y -2667.355,Z 190.712,A -89.99946,B 0.00000,C 180.00000} ; preinsert
  LIN {X -12531.996,Y -2667.355,Z -59.288,A -89.99946,B 0.00000,C 180.00000} ; insert
  LIN {X -12531.996,Y -2667.355,Z -59.288,A -89.99946,B 0.00000,C 180.00000} ; release
  LIN {X -12531.996,Y -2667.355,Z 240.712,A -89.99946,B 0.00000,C 180.00000} ; retreat
  ; Step 1855, bar 810
  LIN {X -12431.996,Y -2667.355,Z 1143.930,A -89.99946,B 0.00000,C 180.00000} ; outside
  LIN {X -12431.996,Y -2667.355,Z 190.712,A -89.99946,B 0.00000,C 180.00000} ; preinsert
  LIN {X -12431.996,Y -2667.355,Z -59.288,A -89.99946,B 0.00000,C 180.00000} ; insert
  LIN {X -12431.996,Y -2667.355,Z -59.288,A -89.99946,B 0.00000,C 180.00000} ; release
  LIN {X -12431.996,Y -2667.355,Z 240.712,A -89.99946,B 0.00000,C 180.00000} ; retreat
  ; Step 1856, bar 808
  LIN {X -12331.996,Y -2667.355,Z 1143.930,A -89.99946,B 0.00000,C 180.00000} ; outside
  LIN {X -12331.996,Y -2667.355,Z 190.712,A -89.99946,B 0.00000,C 180.00000} ; preinsert
  LIN {X -12331.996,Y -2667.355,Z -59.288,A -89.99946,B 0.00000,C 180.00000} ; insert
  LIN {X -12331.996,Y -2667.355,Z -59.288,A -89.99946,B 0.00000,C 180.00000} ; release
  LIN {X -12331.996,Y -2667.355,Z 240.712,A -89.99946,B 0.00000,C 180.00000} ; retreat
  ; Step 1857, bar 806
  LIN {X -12231.996,Y -2667.355,Z 1143.930,A -89.99946,B 0.00000,C 180.00000} ; outside
  LIN {X -12231.996,Y -2667.355,Z 190.712,A -89.99946,B 0.00000,C 180.00000} ; preinsert
  LIN {X -12231.996,Y -2667.355,Z -59.288,A -89.99946,B 0.00000,C 180.00000} ; insert
  LIN {X -12231.996,Y -2667.355,Z -59.288,A -89.99946,B 0.00000,C 180.00000} ; release
  LIN {X -12231.996,Y -2667.355,Z 240.712,A -89.99946,B 0.00000,C 180.00000} ; retreat
  ; Step 1858, bar 804
  LIN {X -12106.996,Y -2667.355,Z 1143.930,A -89.99946,B 0.00000,C 180.00000} ; outside
  LIN {X -12106.996,Y -2667.355,Z 190.712,A -89.99946,B 0.00000,C 180.00000} ; preinsert
  LIN {X -12106.996,Y -2667.355,Z -59.288,A -89.99946,B 0.00000,C 180.00000} ; insert
  LIN {X -12106.996,Y -2667.355,Z -59.288,A -89.99946,B 0.00000,C 180.00000} ; release
  LIN {X -12106.996,Y -2667.355,Z 240.712,A -89.99946,B 0.00000,C 180.00000} ; retreat
  ; Step 1859, bar 802
  LIN {X -11981.996,Y -2667.355,Z 1143.930,A -89.99946,B 0.00000,C 180.00000} ; outside
  LIN {X -11981.996,Y -2667.355,Z 190.712,A -89.99946,B 0.00000,C 180.00000} ; preinsert
  LIN {X -11981.996,Y -2667.355,Z -59.288,A -89.99946,B 0.00000,C 180.00000} ; insert
  LIN {X -11981.996,Y -2667.355,Z -59.288,A -89.99946,B 0.00000,C 180.00000} ; release
  LIN {X -11981.996,Y -2667.355,Z 240.712,A -89.99946,B 0.00000,C 180.00000} ; retreat
  ; Step 1860, bar 800
  LIN {X -11856.996,Y -2667.355,Z 1143.930,A -89.99946,B 0.00000,C 180.00000} ; outside
  LIN {X -11856.996,Y -2667.355,Z 190.712,A -89.99946,B 0.00000,C 180.00000} ; preinsert
  LIN {X -11856.996,Y -2667.355,Z -59.288,A -89.99946,B 0.00000,C 180.00000} ; insert
  LIN {X -11856.996,Y -2667.355,Z -59.288,A -89.99946,B 0.00000,C 180.00000} ; release
  LIN {X -11856.996,Y -2667.355,Z 240.712,A -89.99946,B 0.00000,C 180.00000} ; retreat
  ; Step 1861, bar 798
  LIN {X -11731.996,Y -2667.355,Z 1143.930,A -89.99946,B 0.00000,C 180.00000} ; outside
  LIN {X -11731.996,Y -2667.355,Z 190.712,A -89.99946,B 0.00000,C 180.00000} ; preinsert
  LIN {X -11731.996,Y -2667.355,Z -59.288,A -89.99946,B 0.00000,C 180.00000} ; insert
  LIN {X -11731.996,Y -2667.355,Z -59.288,A -89.99946,B 0.00000,C 180.00000} ; release
  LIN {X -11731.996,Y -2667.355,Z 240.712,A -89.99946,B 0.00000,C 180.00000} ; retreat
  ; Step 1862, bar 796
  LIN {X -11606.996,Y -2667.355,Z 1143.930,A -89.99946,B 0.00000,C 180.00000} ; outside
  LIN {X -11606.996,Y -2667.355,Z 190.712,A -89.99946,B 0.00000,C 180.00000} ; preinsert
  LIN {X -11606.996,Y -2667.355,Z -59.288,A -89.99946,B 0.00000,C 180.00000} ; insert
  LIN {X -11606.996,Y -2667.355,Z -59.288,A -89.99946,B 0.00000,C 180.00000} ; release
  LIN {X -11606.996,Y -2667.355,Z 240.712,A -89.99946,B 0.00000,C 180.00000} ; retreat
  ; Step 1863, bar 794
  LIN {X -11481.996,Y -2667.355,Z 1143.930,A -89.99946,B 0.00000,C 180.00000} ; outside
  LIN {X -11481.996,Y -2667.355,Z 190.712,A -89.99946,B 0.00000,C 180.00000} ; preinsert
  LIN {X -11481.996,Y -2667.355,Z -59.288,A -89.99946,B 0.00000,C 180.00000} ; insert
  LIN {X -11481.996,Y -2667.355,Z -59.288,A -89.99946,B 0.00000,C 180.00000} ; release
  LIN {X -11481.996,Y -2667.355,Z 240.712,A -89.99946,B 0.00000,C 180.00000} ; retreat
  ; Step 1864, bar 792
  LIN {X -11356.996,Y -2667.355,Z 1143.930,A -89.99946,B 0.00000,C 180.00000} ; outside
  LIN {X -11356.996,Y -2667.355,Z 190.712,A -89.99946,B 0.00000,C 180.00000} ; preinsert
  LIN {X -11356.996,Y -2667.355,Z -59.288,A -89.99946,B 0.00000,C 180.00000} ; insert
  LIN {X -11356.996,Y -2667.355,Z -59.288,A -89.99946,B 0.00000,C 180.00000} ; release
  LIN {X -11356.996,Y -2667.355,Z 240.712,A -89.99946,B 0.00000,C 180.00000} ; retreat
  ; Step 1865, bar 790
  LIN {X -11231.996,Y -2667.355,Z 1143.930,A -89.99946,B 0.00000,C 180.00000} ; outside
  LIN {X -11231.996,Y -2667.355,Z 190.712,A -89.99946,B 0.00000,C 180.00000} ; preinsert
  LIN {X -11231.996,Y -2667.355,Z -59.288,A -89.99946,B 0.00000,C 180.00000} ; insert
  LIN {X -11231.996,Y -2667.355,Z -59.288,A -89.99946,B 0.00000,C 180.00000} ; release
  LIN {X -11231.996,Y -2667.355,Z 240.712,A -89.99946,B 0.00000,C 180.00000} ; retreat
  ; Step 1866, bar 788
  LIN {X -11106.996,Y -2667.355,Z 1143.930,A -89.99946,B 0.00000,C 180.00000} ; outside
  LIN {X -11106.996,Y -2667.355,Z 190.712,A -89.99946,B 0.00000,C 180.00000} ; preinsert
  LIN {X -11106.996,Y -2667.355,Z -59.288,A -89.99946,B 0.00000,C 180.00000} ; insert
  LIN {X -11106.996,Y -2667.355,Z -59.288,A -89.99946,B 0.00000,C 180.00000} ; release
  LIN {X -11106.996,Y -2667.355,Z 240.712,A -89.99946,B 0.00000,C 180.00000} ; retreat
  ; Step 1867, bar 786
  LIN {X -10981.996,Y -2667.355,Z 1143.930,A -89.99946,B 0.00000,C 180.00000} ; outside
  LIN {X -10981.996,Y -2667.355,Z 190.712,A -89.99946,B 0.00000,C 180.00000} ; preinsert
  LIN {X -10981.996,Y -2667.355,Z -59.288,A -89.99946,B 0.00000,C 180.00000} ; insert
  LIN {X -10981.996,Y -2667.355,Z -59.288,A -89.99946,B 0.00000,C 180.00000} ; release
  LIN {X -10981.996,Y -2667.355,Z 240.712,A -89.99946,B 0.00000,C 180.00000} ; retreat
  ; Step 1868, bar 784
  LIN {X -10856.996,Y -2667.355,Z 1143.930,A -89.99946,B 0.00000,C 180.00000} ; outside
  LIN {X -10856.996,Y -2667.355,Z 190.712,A -89.99946,B 0.00000,C 180.00000} ; preinsert
  LIN {X -10856.996,Y -2667.355,Z -59.288,A -89.99946,B 0.00000,C 180.00000} ; insert
  LIN {X -10856.996,Y -2667.355,Z -59.288,A -89.99946,B 0.00000,C 180.00000} ; release
  LIN {X -10856.996,Y -2667.355,Z 240.712,A -89.99946,B 0.00000,C 180.00000} ; retreat
  ; Step 1869, bar 782
  LIN {X -10731.996,Y -2667.355,Z 1143.930,A -89.99946,B 0.00000,C 180.00000} ; outside
  LIN {X -10731.996,Y -2667.355,Z 190.712,A -89.99946,B 0.00000,C 180.00000} ; preinsert
  LIN {X -10731.996,Y -2667.355,Z -59.288,A -89.99946,B 0.00000,C 180.00000} ; insert
  LIN {X -10731.996,Y -2667.355,Z -59.288,A -89.99946,B 0.00000,C 180.00000} ; release
  LIN {X -10731.996,Y -2667.355,Z 240.712,A -89.99946,B 0.00000,C 180.00000} ; retreat
  ; Step 1870, bar 780
  LIN {X -10606.996,Y -2667.355,Z 1143.930,A -89.99946,B 0.00000,C 180.00000} ; outside
  LIN {X -10606.996,Y -2667.355,Z 190.712,A -89.99946,B 0.00000,C 180.00000} ; preinsert
  LIN {X -10606.996,Y -2667.355,Z -59.288,A -89.99946,B 0.00000,C 180.00000} ; insert
  LIN {X -10606.996,Y -2667.355,Z -59.288,A -89.99946,B 0.00000,C 180.00000} ; release
  LIN {X -10606.996,Y -2667.355,Z 240.712,A -89.99946,B 0.00000,C 180.00000} ; retreat
  ; Step 1871, bar 778
  LIN {X -10481.996,Y -2667.355,Z 1143.930,A -89.99946,B 0.00000,C 180.00000} ; outside
  LIN {X -10481.996,Y -2667.355,Z 190.712,A -89.99946,B 0.00000,C 180.00000} ; preinsert
  LIN {X -10481.996,Y -2667.355,Z -59.288,A -89.99946,B 0.00000,C 180.00000} ; insert
  LIN {X -10481.996,Y -2667.355,Z -59.288,A -89.99946,B 0.00000,C 180.00000} ; release
  LIN {X -10481.996,Y -2667.355,Z 240.712,A -89.99946,B 0.00000,C 180.00000} ; retreat
  ; Step 1872, bar 776
  LIN {X -10356.996,Y -2667.355,Z 1143.930,A -89.99946,B 0.00000,C 180.00000} ; outside
  LIN {X -10356.996,Y -2667.355,Z 190.712,A -89.99946,B 0.00000,C 180.00000} ; preinsert
  LIN {X -10356.996,Y -2667.355,Z -59.288,A -89.99946,B 0.00000,C 180.00000} ; insert
  LIN {X -10356.996,Y -2667.355,Z -59.288,A -89.99946,B 0.00000,C 180.00000} ; release
  LIN {X -10356.996,Y -2667.355,Z 240.712,A -89.99946,B 0.00000,C 180.00000} ; retreat
  ; Step 1873, bar 774
  LIN {X -10231.996,Y -2667.355,Z 1143.930,A -89.99946,B 0.00000,C 180.00000} ; outside
  LIN {X -10231.996,Y -2667.355,Z 190.712,A -89.99946,B 0.00000,C 180.00000} ; preinsert
  LIN {X -10231.996,Y -2667.355,Z -59.288,A -89.99946,B 0.00000,C 180.00000} ; insert
  LIN {X -10231.996,Y -2667.355,Z -59.288,A -89.99946,B 0.00000,C 180.00000} ; release
  LIN {X -10231.996,Y -2667.355,Z 240.712,A -89.99946,B 0.00000,C 180.00000} ; retreat
  ; Step 1874, bar 772
  LIN {X -10106.996,Y -2667.355,Z 1143.930,A -89.99946,B 0.00000,C 180.00000} ; outside
  LIN {X -10106.996,Y -2667.355,Z 190.712,A -89.99946,B 0.00000,C 180.00000} ; preinsert
  LIN {X -10106.996,Y -2667.355,Z -59.288,A -89.99946,B 0.00000,C 180.00000} ; insert
  LIN {X -10106.996,Y -2667.355,Z -59.288,A -89.99946,B 0.00000,C 180.00000} ; release
  LIN {X -10106.996,Y -2667.355,Z 240.712,A -89.99946,B 0.00000,C 180.00000} ; retreat
  ; Step 1875, bar 770
  LIN {X -9856.996,Y -2667.355,Z 1143.930,A -89.99946,B 0.00000,C 180.00000} ; outside
  LIN {X -9856.996,Y -2667.355,Z 190.712,A -89.99946,B 0.00000,C 180.00000} ; preinsert
  LIN {X -9856.996,Y -2667.355,Z -59.288,A -89.99946,B 0.00000,C 180.00000} ; insert
  LIN {X -9856.996,Y -2667.355,Z -59.288,A -89.99946,B 0.00000,C 180.00000} ; release
  LIN {X -9856.996,Y -2667.355,Z 240.712,A -89.99946,B 0.00000,C 180.00000} ; retreat
  ; Step 1876, bar 768
  LIN {X -9731.996,Y -2667.355,Z 1143.930,A -89.99946,B 0.00000,C 180.00000} ; outside
  LIN {X -9731.996,Y -2667.355,Z 190.712,A -89.99946,B 0.00000,C 180.00000} ; preinsert
  LIN {X -9731.996,Y -2667.355,Z -59.288,A -89.99946,B 0.00000,C 180.00000} ; insert
  LIN {X -9731.996,Y -2667.355,Z -59.288,A -89.99946,B 0.00000,C 180.00000} ; release
  LIN {X -9731.996,Y -2667.355,Z 240.712,A -89.99946,B 0.00000,C 180.00000} ; retreat
  ; Step 1877, bar 766
  LIN {X -9606.996,Y -2667.355,Z 1143.930,A -89.99946,B 0.00000,C 180.00000} ; outside
  LIN {X -9606.996,Y -2667.355,Z 190.712,A -89.99946,B 0.00000,C 180.00000} ; preinsert
  LIN {X -9606.996,Y -2667.355,Z -59.288,A -89.99946,B 0.00000,C 180.00000} ; insert
  LIN {X -9606.996,Y -2667.355,Z -59.288,A -89.99946,B 0.00000,C 180.00000} ; release
  LIN {X -9606.996,Y -2667.355,Z 240.712,A -89.99946,B 0.00000,C 180.00000} ; retreat
  ; Step 1878, bar 764
  LIN {X -9481.996,Y -2667.355,Z 1143.930,A -89.99946,B 0.00000,C 180.00000} ; outside
  LIN {X -9481.996,Y -2667.355,Z 190.712,A -89.99946,B 0.00000,C 180.00000} ; preinsert
  LIN {X -9481.996,Y -2667.355,Z -59.288,A -89.99946,B 0.00000,C 180.00000} ; insert
  LIN {X -9481.996,Y -2667.355,Z -59.288,A -89.99946,B 0.00000,C 180.00000} ; release
  LIN {X -9481.996,Y -2667.355,Z 240.712,A -89.99946,B 0.00000,C 180.00000} ; retreat
  ; Step 1879, bar 762
  LIN {X -9356.996,Y -2667.355,Z 1143.930,A -89.99946,B 0.00000,C 180.00000} ; outside
  LIN {X -9356.996,Y -2667.355,Z 190.712,A -89.99946,B 0.00000,C 180.00000} ; preinsert
  LIN {X -9356.996,Y -2667.355,Z -59.288,A -89.99946,B 0.00000,C 180.00000} ; insert
  LIN {X -9356.996,Y -2667.355,Z -59.288,A -89.99946,B 0.00000,C 180.00000} ; release
  LIN {X -9356.996,Y -2667.355,Z 240.712,A -89.99946,B 0.00000,C 180.00000} ; retreat
  ; Step 1880, bar 760
  LIN {X -9231.996,Y -2667.355,Z 1143.930,A -89.99946,B 0.00000,C 180.00000} ; outside
  LIN {X -9231.996,Y -2667.355,Z 190.712,A -89.99946,B 0.00000,C 180.00000} ; preinsert
  LIN {X -9231.996,Y -2667.355,Z -59.288,A -89.99946,B 0.00000,C 180.00000} ; insert
  LIN {X -9231.996,Y -2667.355,Z -59.288,A -89.99946,B 0.00000,C 180.00000} ; release
  LIN {X -9231.996,Y -2667.355,Z 240.712,A -89.99946,B 0.00000,C 180.00000} ; retreat
  ; Step 1881, bar 758
  LIN {X -9106.996,Y -2667.355,Z 1143.930,A -89.99946,B 0.00000,C 180.00000} ; outside
  LIN {X -9106.996,Y -2667.355,Z 190.712,A -89.99946,B 0.00000,C 180.00000} ; preinsert
  LIN {X -9106.996,Y -2667.355,Z -59.288,A -89.99946,B 0.00000,C 180.00000} ; insert
  LIN {X -9106.996,Y -2667.355,Z -59.288,A -89.99946,B 0.00000,C 180.00000} ; release
  LIN {X -9106.996,Y -2667.355,Z 240.712,A -89.99946,B 0.00000,C 180.00000} ; retreat
  ; Step 1882, bar 756
  LIN {X -8981.996,Y -2667.355,Z 1143.930,A -89.99946,B 0.00000,C 180.00000} ; outside
  LIN {X -8981.996,Y -2667.355,Z 190.712,A -89.99946,B 0.00000,C 180.00000} ; preinsert
  LIN {X -8981.996,Y -2667.355,Z -59.288,A -89.99946,B 0.00000,C 180.00000} ; insert
  LIN {X -8981.996,Y -2667.355,Z -59.288,A -89.99946,B 0.00000,C 180.00000} ; release
  LIN {X -8981.996,Y -2667.355,Z 240.712,A -89.99946,B 0.00000,C 180.00000} ; retreat
  ; Step 1883, bar 754
  LIN {X -8856.996,Y -2667.355,Z 1143.930,A -89.99946,B 0.00000,C 180.00000} ; outside
  LIN {X -8856.996,Y -2667.355,Z 190.712,A -89.99946,B 0.00000,C 180.00000} ; preinsert
  LIN {X -8856.996,Y -2667.355,Z -59.288,A -89.99946,B 0.00000,C 180.00000} ; insert
  LIN {X -8856.996,Y -2667.355,Z -59.288,A -89.99946,B 0.00000,C 180.00000} ; release
  LIN {X -8856.996,Y -2667.355,Z 240.712,A -89.99946,B 0.00000,C 180.00000} ; retreat
  ; Step 1884, bar 752
  LIN {X -8731.996,Y -2667.355,Z 1143.930,A -89.99946,B 0.00000,C 180.00000} ; outside
  LIN {X -8731.996,Y -2667.355,Z 190.712,A -89.99946,B 0.00000,C 180.00000} ; preinsert
  LIN {X -8731.996,Y -2667.355,Z -59.288,A -89.99946,B 0.00000,C 180.00000} ; insert
  LIN {X -8731.996,Y -2667.355,Z -59.288,A -89.99946,B 0.00000,C 180.00000} ; release
  LIN {X -8731.996,Y -2667.355,Z 240.712,A -89.99946,B 0.00000,C 180.00000} ; retreat
  ; Step 1885, bar 750
  LIN {X -8606.996,Y -2667.355,Z 1143.930,A -89.99946,B 0.00000,C 180.00000} ; outside
  LIN {X -8606.996,Y -2667.355,Z 190.712,A -89.99946,B 0.00000,C 180.00000} ; preinsert
  LIN {X -8606.996,Y -2667.355,Z -59.288,A -89.99946,B 0.00000,C 180.00000} ; insert
  LIN {X -8606.996,Y -2667.355,Z -59.288,A -89.99946,B 0.00000,C 180.00000} ; release
  LIN {X -8606.996,Y -2667.355,Z 240.712,A -89.99946,B 0.00000,C 180.00000} ; retreat
  ; Step 1886, bar 748
  LIN {X -8481.996,Y -2667.355,Z 1143.930,A -89.99946,B 0.00000,C 180.00000} ; outside
  LIN {X -8481.996,Y -2667.355,Z 190.712,A -89.99946,B 0.00000,C 180.00000} ; preinsert
  LIN {X -8481.996,Y -2667.355,Z -59.288,A -89.99946,B 0.00000,C 180.00000} ; insert
  LIN {X -8481.996,Y -2667.355,Z -59.288,A -89.99946,B 0.00000,C 180.00000} ; release
  LIN {X -8481.996,Y -2667.355,Z 240.712,A -89.99946,B 0.00000,C 180.00000} ; retreat
  ; Step 1887, bar 746
  LIN {X -8356.996,Y -2667.355,Z 1143.930,A -89.99946,B 0.00000,C 180.00000} ; outside
  LIN {X -8356.996,Y -2667.355,Z 190.712,A -89.99946,B 0.00000,C 180.00000} ; preinsert
  LIN {X -8356.996,Y -2667.355,Z -59.288,A -89.99946,B 0.00000,C 180.00000} ; insert
  LIN {X -8356.996,Y -2667.355,Z -59.288,A -89.99946,B 0.00000,C 180.00000} ; release
  LIN {X -8356.996,Y -2667.355,Z 240.712,A -89.99946,B 0.00000,C 180.00000} ; retreat
  ; Step 1888, bar 744
  LIN {X -8231.996,Y -2667.355,Z 1143.930,A -89.99946,B 0.00000,C 180.00000} ; outside
  LIN {X -8231.996,Y -2667.355,Z 190.712,A -89.99946,B 0.00000,C 180.00000} ; preinsert
  LIN {X -8231.996,Y -2667.355,Z -59.288,A -89.99946,B 0.00000,C 180.00000} ; insert
  LIN {X -8231.996,Y -2667.355,Z -59.288,A -89.99946,B 0.00000,C 180.00000} ; release
  LIN {X -8231.996,Y -2667.355,Z 240.712,A -89.99946,B 0.00000,C 180.00000} ; retreat
  ; Step 1889, bar 742
  LIN {X -8106.996,Y -2667.355,Z 1143.930,A -89.99946,B 0.00000,C 180.00000} ; outside
  LIN {X -8106.996,Y -2667.355,Z 190.712,A -89.99946,B 0.00000,C 180.00000} ; preinsert
  LIN {X -8106.996,Y -2667.355,Z -59.288,A -89.99946,B 0.00000,C 180.00000} ; insert
  LIN {X -8106.996,Y -2667.355,Z -59.288,A -89.99946,B 0.00000,C 180.00000} ; release
  LIN {X -8106.996,Y -2667.355,Z 240.712,A -89.99946,B 0.00000,C 180.00000} ; retreat
  ; Step 1890, bar 740
  LIN {X -7981.996,Y -2667.355,Z 1143.930,A -89.99946,B 0.00000,C 180.00000} ; outside
  LIN {X -7981.996,Y -2667.355,Z 190.712,A -89.99946,B 0.00000,C 180.00000} ; preinsert
  LIN {X -7981.996,Y -2667.355,Z -59.288,A -89.99946,B 0.00000,C 180.00000} ; insert
  LIN {X -7981.996,Y -2667.355,Z -59.288,A -89.99946,B 0.00000,C 180.00000} ; release
  LIN {X -7981.996,Y -2667.355,Z 240.712,A -89.99946,B 0.00000,C 180.00000} ; retreat
  ; Step 1891, bar 738
  LIN {X -7856.996,Y -2667.355,Z 1143.930,A -89.99946,B 0.00000,C 180.00000} ; outside
  LIN {X -7856.996,Y -2667.355,Z 190.712,A -89.99946,B 0.00000,C 180.00000} ; preinsert
  LIN {X -7856.996,Y -2667.355,Z -59.288,A -89.99946,B 0.00000,C 180.00000} ; insert
  LIN {X -7856.996,Y -2667.355,Z -59.288,A -89.99946,B 0.00000,C 180.00000} ; release
  LIN {X -7856.996,Y -2667.355,Z 240.712,A -89.99946,B 0.00000,C 180.00000} ; retreat
  ; Step 1892, bar 736
  LIN {X -7731.996,Y -2667.355,Z 1143.930,A -89.99946,B 0.00000,C 180.00000} ; outside
  LIN {X -7731.996,Y -2667.355,Z 190.712,A -89.99946,B 0.00000,C 180.00000} ; preinsert
  LIN {X -7731.996,Y -2667.355,Z -59.288,A -89.99946,B 0.00000,C 180.00000} ; insert
  LIN {X -7731.996,Y -2667.355,Z -59.288,A -89.99946,B 0.00000,C 180.00000} ; release
  LIN {X -7731.996,Y -2667.355,Z 240.712,A -89.99946,B 0.00000,C 180.00000} ; retreat
  ; Step 1893, bar 734
  LIN {X -7606.996,Y -2667.355,Z 1143.930,A -89.99946,B 0.00000,C 180.00000} ; outside
  LIN {X -7606.996,Y -2667.355,Z 190.712,A -89.99946,B 0.00000,C 180.00000} ; preinsert
  LIN {X -7606.996,Y -2667.355,Z -59.288,A -89.99946,B 0.00000,C 180.00000} ; insert
  LIN {X -7606.996,Y -2667.355,Z -59.288,A -89.99946,B 0.00000,C 180.00000} ; release
  LIN {X -7606.996,Y -2667.355,Z 240.712,A -89.99946,B 0.00000,C 180.00000} ; retreat
  ; Step 1894, bar 732
  LIN {X -7481.996,Y -2667.355,Z 1143.930,A -89.99946,B 0.00000,C 180.00000} ; outside
  LIN {X -7481.996,Y -2667.355,Z 190.712,A -89.99946,B 0.00000,C 180.00000} ; preinsert
  LIN {X -7481.996,Y -2667.355,Z -59.288,A -89.99946,B 0.00000,C 180.00000} ; insert
  LIN {X -7481.996,Y -2667.355,Z -59.288,A -89.99946,B 0.00000,C 180.00000} ; release
  LIN {X -7481.996,Y -2667.355,Z 240.712,A -89.99946,B 0.00000,C 180.00000} ; retreat
  ; Step 1895, bar 730
  LIN {X -7356.996,Y -2667.355,Z 1143.930,A -89.99946,B 0.00000,C 180.00000} ; outside
  LIN {X -7356.996,Y -2667.355,Z 190.712,A -89.99946,B 0.00000,C 180.00000} ; preinsert
  LIN {X -7356.996,Y -2667.355,Z -59.288,A -89.99946,B 0.00000,C 180.00000} ; insert
  LIN {X -7356.996,Y -2667.355,Z -59.288,A -89.99946,B 0.00000,C 180.00000} ; release
  LIN {X -7356.996,Y -2667.355,Z 240.712,A -89.99946,B 0.00000,C 180.00000} ; retreat
  ; Step 1896, bar 728
  LIN {X -7231.996,Y -2667.355,Z 1143.930,A -89.99946,B 0.00000,C 180.00000} ; outside
  LIN {X -7231.996,Y -2667.355,Z 190.712,A -89.99946,B 0.00000,C 180.00000} ; preinsert
  LIN {X -7231.996,Y -2667.355,Z -59.288,A -89.99946,B 0.00000,C 180.00000} ; insert
  LIN {X -7231.996,Y -2667.355,Z -59.288,A -89.99946,B 0.00000,C 180.00000} ; release
  LIN {X -7231.996,Y -2667.355,Z 240.712,A -89.99946,B 0.00000,C 180.00000} ; retreat
  ; Step 1897, bar 726
  LIN {X -7106.996,Y -2667.355,Z 1143.930,A -89.99946,B 0.00000,C 180.00000} ; outside
  LIN {X -7106.996,Y -2667.355,Z 190.712,A -89.99946,B 0.00000,C 180.00000} ; preinsert
  LIN {X -7106.996,Y -2667.355,Z -59.288,A -89.99946,B 0.00000,C 180.00000} ; insert
  LIN {X -7106.996,Y -2667.355,Z -59.288,A -89.99946,B 0.00000,C 180.00000} ; release
  LIN {X -7106.996,Y -2667.355,Z 240.712,A -89.99946,B 0.00000,C 180.00000} ; retreat
  ; Step 1898, bar 724
  LIN {X -6981.996,Y -2667.355,Z 1143.930,A -89.99946,B 0.00000,C 180.00000} ; outside
  LIN {X -6981.996,Y -2667.355,Z 190.712,A -89.99946,B 0.00000,C 180.00000} ; preinsert
  LIN {X -6981.996,Y -2667.355,Z -59.288,A -89.99946,B 0.00000,C 180.00000} ; insert
  LIN {X -6981.996,Y -2667.355,Z -59.288,A -89.99946,B 0.00000,C 180.00000} ; release
  LIN {X -6981.996,Y -2667.355,Z 240.712,A -89.99946,B 0.00000,C 180.00000} ; retreat
  ; Step 1899, bar 722
  LIN {X -6856.996,Y -2667.355,Z 1143.930,A -89.99946,B 0.00000,C 180.00000} ; outside
  LIN {X -6856.996,Y -2667.355,Z 190.712,A -89.99946,B 0.00000,C 180.00000} ; preinsert
  LIN {X -6856.996,Y -2667.355,Z -59.288,A -89.99946,B 0.00000,C 180.00000} ; insert
  LIN {X -6856.996,Y -2667.355,Z -59.288,A -89.99946,B 0.00000,C 180.00000} ; release
  LIN {X -6856.996,Y -2667.355,Z 240.712,A -89.99946,B 0.00000,C 180.00000} ; retreat
  ; Step 1900, bar 720
  LIN {X -6731.996,Y -2667.355,Z 1143.930,A -89.99946,B 0.00000,C 180.00000} ; outside
  LIN {X -6731.996,Y -2667.355,Z 190.712,A -89.99946,B 0.00000,C 180.00000} ; preinsert
  LIN {X -6731.996,Y -2667.355,Z -59.288,A -89.99946,B 0.00000,C 180.00000} ; insert
  LIN {X -6731.996,Y -2667.355,Z -59.288,A -89.99946,B 0.00000,C 180.00000} ; release
  LIN {X -6731.996,Y -2667.355,Z 240.712,A -89.99946,B 0.00000,C 180.00000} ; retreat
  ; Step 1901, bar 718
  LIN {X -6606.996,Y -2667.355,Z 1143.930,A -89.99946,B 0.00000,C 180.00000} ; outside
  LIN {X -6606.996,Y -2667.355,Z 190.712,A -89.99946,B 0.00000,C 180.00000} ; preinsert
  LIN {X -6606.996,Y -2667.355,Z -59.288,A -89.99946,B 0.00000,C 180.00000} ; insert
  LIN {X -6606.996,Y -2667.355,Z -59.288,A -89.99946,B 0.00000,C 180.00000} ; release
  LIN {X -6606.996,Y -2667.355,Z 240.712,A -89.99946,B 0.00000,C 180.00000} ; retreat
  ; Step 1902, bar 716
  LIN {X -6481.996,Y -2667.355,Z 1143.930,A -89.99946,B 0.00000,C 180.00000} ; outside
  LIN {X -6481.996,Y -2667.355,Z 190.712,A -89.99946,B 0.00000,C 180.00000} ; preinsert
  LIN {X -6481.996,Y -2667.355,Z -59.288,A -89.99946,B 0.00000,C 180.00000} ; insert
  LIN {X -6481.996,Y -2667.355,Z -59.288,A -89.99946,B 0.00000,C 180.00000} ; release
  LIN {X -6481.996,Y -2667.355,Z 240.712,A -89.99946,B 0.00000,C 180.00000} ; retreat
  ; Step 1903, bar 714
  LIN {X -6356.996,Y -2667.355,Z 1143.930,A -89.99946,B 0.00000,C 180.00000} ; outside
  LIN {X -6356.996,Y -2667.355,Z 190.712,A -89.99946,B 0.00000,C 180.00000} ; preinsert
  LIN {X -6356.996,Y -2667.355,Z -59.288,A -89.99946,B 0.00000,C 180.00000} ; insert
  LIN {X -6356.996,Y -2667.355,Z -59.288,A -89.99946,B 0.00000,C 180.00000} ; release
  LIN {X -6356.996,Y -2667.355,Z 240.712,A -89.99946,B 0.00000,C 180.00000} ; retreat
  ; Step 1904, bar 712
  LIN {X -6231.996,Y -2667.355,Z 1143.930,A -89.99946,B 0.00000,C 180.00000} ; outside
  LIN {X -6231.996,Y -2667.355,Z 190.712,A -89.99946,B 0.00000,C 180.00000} ; preinsert
  LIN {X -6231.996,Y -2667.355,Z -59.288,A -89.99946,B 0.00000,C 180.00000} ; insert
  LIN {X -6231.996,Y -2667.355,Z -59.288,A -89.99946,B 0.00000,C 180.00000} ; release
  LIN {X -6231.996,Y -2667.355,Z 240.712,A -89.99946,B 0.00000,C 180.00000} ; retreat
  ; Step 1905, bar 710
  LIN {X -6106.996,Y -2667.355,Z 1143.930,A -89.99946,B 0.00000,C 180.00000} ; outside
  LIN {X -6106.996,Y -2667.355,Z 190.712,A -89.99946,B 0.00000,C 180.00000} ; preinsert
  LIN {X -6106.996,Y -2667.355,Z -59.288,A -89.99946,B 0.00000,C 180.00000} ; insert
  LIN {X -6106.996,Y -2667.355,Z -59.288,A -89.99946,B 0.00000,C 180.00000} ; release
  LIN {X -6106.996,Y -2667.355,Z 240.712,A -89.99946,B 0.00000,C 180.00000} ; retreat
  ; Step 1906, bar 708
  LIN {X -5856.996,Y -2667.355,Z 1143.930,A -89.99946,B 0.00000,C 180.00000} ; outside
  LIN {X -5856.996,Y -2667.355,Z 190.712,A -89.99946,B 0.00000,C 180.00000} ; preinsert
  LIN {X -5856.996,Y -2667.355,Z -59.288,A -89.99946,B 0.00000,C 180.00000} ; insert
  LIN {X -5856.996,Y -2667.355,Z -59.288,A -89.99946,B 0.00000,C 180.00000} ; release
  LIN {X -5856.996,Y -2667.355,Z 240.712,A -89.99946,B 0.00000,C 180.00000} ; retreat
  ; Step 1907, bar 706
  LIN {X -5731.996,Y -2667.355,Z 1143.930,A -89.99946,B 0.00000,C 180.00000} ; outside
  LIN {X -5731.996,Y -2667.355,Z 190.712,A -89.99946,B 0.00000,C 180.00000} ; preinsert
  LIN {X -5731.996,Y -2667.355,Z -59.288,A -89.99946,B 0.00000,C 180.00000} ; insert
  LIN {X -5731.996,Y -2667.355,Z -59.288,A -89.99946,B 0.00000,C 180.00000} ; release
  LIN {X -5731.996,Y -2667.355,Z 240.712,A -89.99946,B 0.00000,C 180.00000} ; retreat
  ; Step 1908, bar 704
  LIN {X -5606.996,Y -2667.355,Z 1143.930,A -89.99946,B 0.00000,C 180.00000} ; outside
  LIN {X -5606.996,Y -2667.355,Z 190.712,A -89.99946,B 0.00000,C 180.00000} ; preinsert
  LIN {X -5606.996,Y -2667.355,Z -59.288,A -89.99946,B 0.00000,C 180.00000} ; insert
  LIN {X -5606.996,Y -2667.355,Z -59.288,A -89.99946,B 0.00000,C 180.00000} ; release
  LIN {X -5606.996,Y -2667.355,Z 240.712,A -89.99946,B 0.00000,C 180.00000} ; retreat
  ; Step 1909, bar 702
  LIN {X -5481.996,Y -2667.355,Z 1143.930,A -89.99946,B 0.00000,C 180.00000} ; outside
  LIN {X -5481.996,Y -2667.355,Z 190.712,A -89.99946,B 0.00000,C 180.00000} ; preinsert
  LIN {X -5481.996,Y -2667.355,Z -59.288,A -89.99946,B 0.00000,C 180.00000} ; insert
  LIN {X -5481.996,Y -2667.355,Z -59.288,A -89.99946,B 0.00000,C 180.00000} ; release
  LIN {X -5481.996,Y -2667.355,Z 240.712,A -89.99946,B 0.00000,C 180.00000} ; retreat
  ; Step 1910, bar 700
  LIN {X -5356.996,Y -2667.355,Z 1143.930,A -89.99946,B 0.00000,C 180.00000} ; outside
  LIN {X -5356.996,Y -2667.355,Z 190.712,A -89.99946,B 0.00000,C 180.00000} ; preinsert
  LIN {X -5356.996,Y -2667.355,Z -59.288,A -89.99946,B 0.00000,C 180.00000} ; insert
  LIN {X -5356.996,Y -2667.355,Z -59.288,A -89.99946,B 0.00000,C 180.00000} ; release
  LIN {X -5356.996,Y -2667.355,Z 240.712,A -89.99946,B 0.00000,C 180.00000} ; retreat
  ; Step 1911, bar 698
  LIN {X -5231.996,Y -2667.355,Z 1143.930,A -89.99946,B 0.00000,C 180.00000} ; outside
  LIN {X -5231.996,Y -2667.355,Z 190.712,A -89.99946,B 0.00000,C 180.00000} ; preinsert
  LIN {X -5231.996,Y -2667.355,Z -59.288,A -89.99946,B 0.00000,C 180.00000} ; insert
  LIN {X -5231.996,Y -2667.355,Z -59.288,A -89.99946,B 0.00000,C 180.00000} ; release
  LIN {X -5231.996,Y -2667.355,Z 240.712,A -89.99946,B 0.00000,C 180.00000} ; retreat
  ; Step 1912, bar 696
  LIN {X -5106.996,Y -2667.355,Z 1143.930,A -89.99946,B 0.00000,C 180.00000} ; outside
  LIN {X -5106.996,Y -2667.355,Z 190.712,A -89.99946,B 0.00000,C 180.00000} ; preinsert
  LIN {X -5106.996,Y -2667.355,Z -59.288,A -89.99946,B 0.00000,C 180.00000} ; insert
  LIN {X -5106.996,Y -2667.355,Z -59.288,A -89.99946,B 0.00000,C 180.00000} ; release
  LIN {X -5106.996,Y -2667.355,Z 240.712,A -89.99946,B 0.00000,C 180.00000} ; retreat
  ; Step 1913, bar 694
  LIN {X -4981.996,Y -2667.355,Z 1143.930,A -89.99946,B 0.00000,C 180.00000} ; outside
  LIN {X -4981.996,Y -2667.355,Z 190.712,A -89.99946,B 0.00000,C 180.00000} ; preinsert
  LIN {X -4981.996,Y -2667.355,Z -59.288,A -89.99946,B 0.00000,C 180.00000} ; insert
  LIN {X -4981.996,Y -2667.355,Z -59.288,A -89.99946,B 0.00000,C 180.00000} ; release
  LIN {X -4981.996,Y -2667.355,Z 240.712,A -89.99946,B 0.00000,C 180.00000} ; retreat
  ; Step 1914, bar 692
  LIN {X -4856.996,Y -2667.355,Z 1143.930,A -89.99946,B 0.00000,C 180.00000} ; outside
  LIN {X -4856.996,Y -2667.355,Z 190.712,A -89.99946,B 0.00000,C 180.00000} ; preinsert
  LIN {X -4856.996,Y -2667.355,Z -59.288,A -89.99946,B 0.00000,C 180.00000} ; insert
  LIN {X -4856.996,Y -2667.355,Z -59.288,A -89.99946,B 0.00000,C 180.00000} ; release
  LIN {X -4856.996,Y -2667.355,Z 240.712,A -89.99946,B 0.00000,C 180.00000} ; retreat
  ; Step 1915, bar 690
  LIN {X -4731.996,Y -2667.355,Z 1143.930,A -89.99946,B 0.00000,C 180.00000} ; outside
  LIN {X -4731.996,Y -2667.355,Z 190.712,A -89.99946,B 0.00000,C 180.00000} ; preinsert
  LIN {X -4731.996,Y -2667.355,Z -59.288,A -89.99946,B 0.00000,C 180.00000} ; insert
  LIN {X -4731.996,Y -2667.355,Z -59.288,A -89.99946,B 0.00000,C 180.00000} ; release
  LIN {X -4731.996,Y -2667.355,Z 240.712,A -89.99946,B 0.00000,C 180.00000} ; retreat
  ; Step 1916, bar 688
  LIN {X -4606.996,Y -2667.355,Z 1143.930,A -89.99946,B 0.00000,C 180.00000} ; outside
  LIN {X -4606.996,Y -2667.355,Z 190.712,A -89.99946,B 0.00000,C 180.00000} ; preinsert
  LIN {X -4606.996,Y -2667.355,Z -59.288,A -89.99946,B 0.00000,C 180.00000} ; insert
  LIN {X -4606.996,Y -2667.355,Z -59.288,A -89.99946,B 0.00000,C 180.00000} ; release
  LIN {X -4606.996,Y -2667.355,Z 240.712,A -89.99946,B 0.00000,C 180.00000} ; retreat
  ; Step 1917, bar 686
  LIN {X -4481.996,Y -2667.355,Z 1143.930,A -89.99946,B 0.00000,C 180.00000} ; outside
  LIN {X -4481.996,Y -2667.355,Z 190.712,A -89.99946,B 0.00000,C 180.00000} ; preinsert
  LIN {X -4481.996,Y -2667.355,Z -59.288,A -89.99946,B 0.00000,C 180.00000} ; insert
  LIN {X -4481.996,Y -2667.355,Z -59.288,A -89.99946,B 0.00000,C 180.00000} ; release
  LIN {X -4481.996,Y -2667.355,Z 240.712,A -89.99946,B 0.00000,C 180.00000} ; retreat
  ; Step 1918, bar 684
  LIN {X -4356.996,Y -2667.355,Z 1143.930,A -89.99946,B 0.00000,C 180.00000} ; outside
  LIN {X -4356.996,Y -2667.355,Z 190.712,A -89.99946,B 0.00000,C 180.00000} ; preinsert
  LIN {X -4356.996,Y -2667.355,Z -59.288,A -89.99946,B 0.00000,C 180.00000} ; insert
  LIN {X -4356.996,Y -2667.355,Z -59.288,A -89.99946,B 0.00000,C 180.00000} ; release
  LIN {X -4356.996,Y -2667.355,Z 240.712,A -89.99946,B 0.00000,C 180.00000} ; retreat
  ; Step 1919, bar 682
  LIN {X -4231.996,Y -2667.355,Z 1143.930,A -89.99946,B 0.00000,C 180.00000} ; outside
  LIN {X -4231.996,Y -2667.355,Z 190.712,A -89.99946,B 0.00000,C 180.00000} ; preinsert
  LIN {X -4231.996,Y -2667.355,Z -59.288,A -89.99946,B 0.00000,C 180.00000} ; insert
  LIN {X -4231.996,Y -2667.355,Z -59.288,A -89.99946,B 0.00000,C 180.00000} ; release
  LIN {X -4231.996,Y -2667.355,Z 240.712,A -89.99946,B 0.00000,C 180.00000} ; retreat
  ; Step 1920, bar 680
  LIN {X -4106.996,Y -2667.355,Z 1143.930,A -89.99946,B 0.00000,C 180.00000} ; outside
  LIN {X -4106.996,Y -2667.355,Z 190.712,A -89.99946,B 0.00000,C 180.00000} ; preinsert
  LIN {X -4106.996,Y -2667.355,Z -59.288,A -89.99946,B 0.00000,C 180.00000} ; insert
  LIN {X -4106.996,Y -2667.355,Z -59.288,A -89.99946,B 0.00000,C 180.00000} ; release
  LIN {X -4106.996,Y -2667.355,Z 240.712,A -89.99946,B 0.00000,C 180.00000} ; retreat
  ; Step 1921, bar 678
  LIN {X -3981.996,Y -2667.355,Z 1143.930,A -89.99946,B 0.00000,C 180.00000} ; outside
  LIN {X -3981.996,Y -2667.355,Z 190.712,A -89.99946,B 0.00000,C 180.00000} ; preinsert
  LIN {X -3981.996,Y -2667.355,Z -59.288,A -89.99946,B 0.00000,C 180.00000} ; insert
  LIN {X -3981.996,Y -2667.355,Z -59.288,A -89.99946,B 0.00000,C 180.00000} ; release
  LIN {X -3981.996,Y -2667.355,Z 240.712,A -89.99946,B 0.00000,C 180.00000} ; retreat
  ; Step 1922, bar 676
  LIN {X -3856.996,Y -2667.355,Z 1143.930,A -89.99946,B 0.00000,C 180.00000} ; outside
  LIN {X -3856.996,Y -2667.355,Z 190.712,A -89.99946,B 0.00000,C 180.00000} ; preinsert
  LIN {X -3856.996,Y -2667.355,Z -59.288,A -89.99946,B 0.00000,C 180.00000} ; insert
  LIN {X -3856.996,Y -2667.355,Z -59.288,A -89.99946,B 0.00000,C 180.00000} ; release
  LIN {X -3856.996,Y -2667.355,Z 240.712,A -89.99946,B 0.00000,C 180.00000} ; retreat
  ; Step 1923, bar 674
  LIN {X -3731.996,Y -2667.355,Z 1143.930,A -89.99946,B 0.00000,C 180.00000} ; outside
  LIN {X -3731.996,Y -2667.355,Z 190.712,A -89.99946,B 0.00000,C 180.00000} ; preinsert
  LIN {X -3731.996,Y -2667.355,Z -59.288,A -89.99946,B 0.00000,C 180.00000} ; insert
  LIN {X -3731.996,Y -2667.355,Z -59.288,A -89.99946,B 0.00000,C 180.00000} ; release
  LIN {X -3731.996,Y -2667.355,Z 240.712,A -89.99946,B 0.00000,C 180.00000} ; retreat
  ; Step 1924, bar 672
  LIN {X -3606.996,Y -2667.355,Z 1143.930,A -89.99946,B 0.00000,C 180.00000} ; outside
  LIN {X -3606.996,Y -2667.355,Z 190.712,A -89.99946,B 0.00000,C 180.00000} ; preinsert
  LIN {X -3606.996,Y -2667.355,Z -59.288,A -89.99946,B 0.00000,C 180.00000} ; insert
  LIN {X -3606.996,Y -2667.355,Z -59.288,A -89.99946,B 0.00000,C 180.00000} ; release
  LIN {X -3606.996,Y -2667.355,Z 240.712,A -89.99946,B 0.00000,C 180.00000} ; retreat
  ; Step 1925, bar 670
  LIN {X -3481.996,Y -2667.355,Z 1143.930,A -89.99946,B 0.00000,C 180.00000} ; outside
  LIN {X -3481.996,Y -2667.355,Z 190.712,A -89.99946,B 0.00000,C 180.00000} ; preinsert
  LIN {X -3481.996,Y -2667.355,Z -59.288,A -89.99946,B 0.00000,C 180.00000} ; insert
  LIN {X -3481.996,Y -2667.355,Z -59.288,A -89.99946,B 0.00000,C 180.00000} ; release
  LIN {X -3481.996,Y -2667.355,Z 240.712,A -89.99946,B 0.00000,C 180.00000} ; retreat
  ; Step 1926, bar 668
  LIN {X -3356.996,Y -2667.355,Z 1143.930,A -89.99946,B 0.00000,C 180.00000} ; outside
  LIN {X -3356.996,Y -2667.355,Z 190.712,A -89.99946,B 0.00000,C 180.00000} ; preinsert
  LIN {X -3356.996,Y -2667.355,Z -59.288,A -89.99946,B 0.00000,C 180.00000} ; insert
  LIN {X -3356.996,Y -2667.355,Z -59.288,A -89.99946,B 0.00000,C 180.00000} ; release
  LIN {X -3356.996,Y -2667.355,Z 240.712,A -89.99946,B 0.00000,C 180.00000} ; retreat
  ; Step 1927, bar 666
  LIN {X -3231.996,Y -2667.355,Z 1143.930,A -89.99946,B 0.00000,C 180.00000} ; outside
  LIN {X -3231.996,Y -2667.355,Z 190.712,A -89.99946,B 0.00000,C 180.00000} ; preinsert
  LIN {X -3231.996,Y -2667.355,Z -59.288,A -89.99946,B 0.00000,C 180.00000} ; insert
  LIN {X -3231.996,Y -2667.355,Z -59.288,A -89.99946,B 0.00000,C 180.00000} ; release
  LIN {X -3231.996,Y -2667.355,Z 240.712,A -89.99946,B 0.00000,C 180.00000} ; retreat
  ; Step 1928, bar 664
  LIN {X -3106.996,Y -2667.355,Z 1143.930,A -89.99946,B 0.00000,C 180.00000} ; outside
  LIN {X -3106.996,Y -2667.355,Z 190.712,A -89.99946,B 0.00000,C 180.00000} ; preinsert
  LIN {X -3106.996,Y -2667.355,Z -59.288,A -89.99946,B 0.00000,C 180.00000} ; insert
  LIN {X -3106.996,Y -2667.355,Z -59.288,A -89.99946,B 0.00000,C 180.00000} ; release
  LIN {X -3106.996,Y -2667.355,Z 240.712,A -89.99946,B 0.00000,C 180.00000} ; retreat
  ; Step 1929, bar 662
  LIN {X -2981.996,Y -2667.355,Z 1143.930,A -89.99946,B 0.00000,C 180.00000} ; outside
  LIN {X -2981.996,Y -2667.355,Z 190.712,A -89.99946,B 0.00000,C 180.00000} ; preinsert
  LIN {X -2981.996,Y -2667.355,Z -59.288,A -89.99946,B 0.00000,C 180.00000} ; insert
  LIN {X -2981.996,Y -2667.355,Z -59.288,A -89.99946,B 0.00000,C 180.00000} ; release
  LIN {X -2981.996,Y -2667.355,Z 240.712,A -89.99946,B 0.00000,C 180.00000} ; retreat
  ; Step 1930, bar 660
  LIN {X -2856.996,Y -2667.355,Z 1143.930,A -89.99946,B 0.00000,C 180.00000} ; outside
  LIN {X -2856.996,Y -2667.355,Z 190.712,A -89.99946,B 0.00000,C 180.00000} ; preinsert
  LIN {X -2856.996,Y -2667.355,Z -59.288,A -89.99946,B 0.00000,C 180.00000} ; insert
  LIN {X -2856.996,Y -2667.355,Z -59.288,A -89.99946,B 0.00000,C 180.00000} ; release
  LIN {X -2856.996,Y -2667.355,Z 240.712,A -89.99946,B 0.00000,C 180.00000} ; retreat
  ; Step 1931, bar 658
  LIN {X -2731.996,Y -2667.355,Z 1143.930,A -89.99946,B 0.00000,C 180.00000} ; outside
  LIN {X -2731.996,Y -2667.355,Z 190.712,A -89.99946,B 0.00000,C 180.00000} ; preinsert
  LIN {X -2731.996,Y -2667.355,Z -59.288,A -89.99946,B 0.00000,C 180.00000} ; insert
  LIN {X -2731.996,Y -2667.355,Z -59.288,A -89.99946,B 0.00000,C 180.00000} ; release
  LIN {X -2731.996,Y -2667.355,Z 240.712,A -89.99946,B 0.00000,C 180.00000} ; retreat
  ; Step 1932, bar 656
  LIN {X -2606.996,Y -2667.355,Z 1143.930,A -89.99946,B 0.00000,C 180.00000} ; outside
  LIN {X -2606.996,Y -2667.355,Z 190.712,A -89.99946,B 0.00000,C 180.00000} ; preinsert
  LIN {X -2606.996,Y -2667.355,Z -59.288,A -89.99946,B 0.00000,C 180.00000} ; insert
  LIN {X -2606.996,Y -2667.355,Z -59.288,A -89.99946,B 0.00000,C 180.00000} ; release
  LIN {X -2606.996,Y -2667.355,Z 240.712,A -89.99946,B 0.00000,C 180.00000} ; retreat
  ; Step 1933, bar 654
  LIN {X -2481.996,Y -2667.355,Z 1143.930,A -89.99946,B 0.00000,C 180.00000} ; outside
  LIN {X -2481.996,Y -2667.355,Z 190.712,A -89.99946,B 0.00000,C 180.00000} ; preinsert
  LIN {X -2481.996,Y -2667.355,Z -59.288,A -89.99946,B 0.00000,C 180.00000} ; insert
  LIN {X -2481.996,Y -2667.355,Z -59.288,A -89.99946,B 0.00000,C 180.00000} ; release
  LIN {X -2481.996,Y -2667.355,Z 240.712,A -89.99946,B 0.00000,C 180.00000} ; retreat
  ; Step 1934, bar 652
  LIN {X -2356.996,Y -2667.355,Z 1143.930,A -89.99946,B 0.00000,C 180.00000} ; outside
  LIN {X -2356.996,Y -2667.355,Z 190.712,A -89.99946,B 0.00000,C 180.00000} ; preinsert
  LIN {X -2356.996,Y -2667.355,Z -59.288,A -89.99946,B 0.00000,C 180.00000} ; insert
  LIN {X -2356.996,Y -2667.355,Z -59.288,A -89.99946,B 0.00000,C 180.00000} ; release
  LIN {X -2356.996,Y -2667.355,Z 240.712,A -89.99946,B 0.00000,C 180.00000} ; retreat
  ; Step 1935, bar 650
  LIN {X -2231.996,Y -2667.355,Z 1143.930,A -89.99946,B 0.00000,C 180.00000} ; outside
  LIN {X -2231.996,Y -2667.355,Z 190.712,A -89.99946,B 0.00000,C 180.00000} ; preinsert
  LIN {X -2231.996,Y -2667.355,Z -59.288,A -89.99946,B 0.00000,C 180.00000} ; insert
  LIN {X -2231.996,Y -2667.355,Z -59.288,A -89.99946,B 0.00000,C 180.00000} ; release
  LIN {X -2231.996,Y -2667.355,Z 240.712,A -89.99946,B 0.00000,C 180.00000} ; retreat
  ; Step 1936, bar 648
  LIN {X -2106.996,Y -2667.355,Z 1143.930,A -89.99946,B 0.00000,C 180.00000} ; outside
  LIN {X -2106.996,Y -2667.355,Z 190.712,A -89.99946,B 0.00000,C 180.00000} ; preinsert
  LIN {X -2106.996,Y -2667.355,Z -59.288,A -89.99946,B 0.00000,C 180.00000} ; insert
  LIN {X -2106.996,Y -2667.355,Z -59.288,A -89.99946,B 0.00000,C 180.00000} ; release
  LIN {X -2106.996,Y -2667.355,Z 240.712,A -89.99946,B 0.00000,C 180.00000} ; retreat
  ; Step 1937, bar 646
  LIN {X -1856.996,Y -2667.355,Z 1143.930,A -89.99946,B 0.00000,C 180.00000} ; outside
  LIN {X -1856.996,Y -2667.355,Z 190.712,A -89.99946,B 0.00000,C 180.00000} ; preinsert
  LIN {X -1856.996,Y -2667.355,Z -59.288,A -89.99946,B 0.00000,C 180.00000} ; insert
  LIN {X -1856.996,Y -2667.355,Z -59.288,A -89.99946,B 0.00000,C 180.00000} ; release
  LIN {X -1856.996,Y -2667.355,Z 240.712,A -89.99946,B 0.00000,C 180.00000} ; retreat
  ; Step 1938, bar 644
  LIN {X -1731.996,Y -2667.355,Z 1143.930,A -89.99946,B 0.00000,C 180.00000} ; outside
  LIN {X -1731.996,Y -2667.355,Z 190.712,A -89.99946,B 0.00000,C 180.00000} ; preinsert
  LIN {X -1731.996,Y -2667.355,Z -59.288,A -89.99946,B 0.00000,C 180.00000} ; insert
  LIN {X -1731.996,Y -2667.355,Z -59.288,A -89.99946,B 0.00000,C 180.00000} ; release
  LIN {X -1731.996,Y -2667.355,Z 240.712,A -89.99946,B 0.00000,C 180.00000} ; retreat
  ; Step 1939, bar 642
  LIN {X -1606.996,Y -2667.355,Z 1143.930,A -89.99946,B 0.00000,C 180.00000} ; outside
  LIN {X -1606.996,Y -2667.355,Z 190.712,A -89.99946,B 0.00000,C 180.00000} ; preinsert
  LIN {X -1606.996,Y -2667.355,Z -59.288,A -89.99946,B 0.00000,C 180.00000} ; insert
  LIN {X -1606.996,Y -2667.355,Z -59.288,A -89.99946,B 0.00000,C 180.00000} ; release
  LIN {X -1606.996,Y -2667.355,Z 240.712,A -89.99946,B 0.00000,C 180.00000} ; retreat
  ; Step 1940, bar 640
  LIN {X -1481.996,Y -2667.355,Z 1143.930,A -89.99946,B 0.00000,C 180.00000} ; outside
  LIN {X -1481.996,Y -2667.355,Z 190.712,A -89.99946,B 0.00000,C 180.00000} ; preinsert
  LIN {X -1481.996,Y -2667.355,Z -59.288,A -89.99946,B 0.00000,C 180.00000} ; insert
  LIN {X -1481.996,Y -2667.355,Z -59.288,A -89.99946,B 0.00000,C 180.00000} ; release
  LIN {X -1481.996,Y -2667.355,Z 240.712,A -89.99946,B 0.00000,C 180.00000} ; retreat
  ; Step 1941, bar 638
  LIN {X -1356.996,Y -2667.355,Z 1143.930,A -89.99946,B 0.00000,C 180.00000} ; outside
  LIN {X -1356.996,Y -2667.355,Z 190.712,A -89.99946,B 0.00000,C 180.00000} ; preinsert
  LIN {X -1356.996,Y -2667.355,Z -59.288,A -89.99946,B 0.00000,C 180.00000} ; insert
  LIN {X -1356.996,Y -2667.355,Z -59.288,A -89.99946,B 0.00000,C 180.00000} ; release
  LIN {X -1356.996,Y -2667.355,Z 240.712,A -89.99946,B 0.00000,C 180.00000} ; retreat
  ; Step 1942, bar 636
  LIN {X -1231.996,Y -2667.355,Z 1143.930,A -89.99946,B 0.00000,C 180.00000} ; outside
  LIN {X -1231.996,Y -2667.355,Z 190.712,A -89.99946,B 0.00000,C 180.00000} ; preinsert
  LIN {X -1231.996,Y -2667.355,Z -59.288,A -89.99946,B 0.00000,C 180.00000} ; insert
  LIN {X -1231.996,Y -2667.355,Z -59.288,A -89.99946,B 0.00000,C 180.00000} ; release
  LIN {X -1231.996,Y -2667.355,Z 240.712,A -89.99946,B 0.00000,C 180.00000} ; retreat
  ; Step 1943, bar 634
  LIN {X -1106.996,Y -2667.355,Z 1143.930,A -89.99946,B 0.00000,C 180.00000} ; outside
  LIN {X -1106.996,Y -2667.355,Z 190.712,A -89.99946,B 0.00000,C 180.00000} ; preinsert
  LIN {X -1106.996,Y -2667.355,Z -59.288,A -89.99946,B 0.00000,C 180.00000} ; insert
  LIN {X -1106.996,Y -2667.355,Z -59.288,A -89.99946,B 0.00000,C 180.00000} ; release
  LIN {X -1106.996,Y -2667.355,Z 240.712,A -89.99946,B 0.00000,C 180.00000} ; retreat
  ; Step 1944, bar 632
  LIN {X -981.996,Y -2667.355,Z 1143.930,A -89.99946,B 0.00000,C 180.00000} ; outside
  LIN {X -981.996,Y -2667.355,Z 190.712,A -89.99946,B 0.00000,C 180.00000} ; preinsert
  LIN {X -981.996,Y -2667.355,Z -59.288,A -89.99946,B 0.00000,C 180.00000} ; insert
  LIN {X -981.996,Y -2667.355,Z -59.288,A -89.99946,B 0.00000,C 180.00000} ; release
  LIN {X -981.996,Y -2667.355,Z 240.712,A -89.99946,B 0.00000,C 180.00000} ; retreat
  ; Step 1945, bar 630
  LIN {X -856.996,Y -2667.355,Z 1143.930,A -89.99946,B 0.00000,C 180.00000} ; outside
  LIN {X -856.996,Y -2667.355,Z 190.712,A -89.99946,B 0.00000,C 180.00000} ; preinsert
  LIN {X -856.996,Y -2667.355,Z -59.288,A -89.99946,B 0.00000,C 180.00000} ; insert
  LIN {X -856.996,Y -2667.355,Z -59.288,A -89.99946,B 0.00000,C 180.00000} ; release
  LIN {X -856.996,Y -2667.355,Z 240.712,A -89.99946,B 0.00000,C 180.00000} ; retreat
  ; Step 1946, bar 628
  LIN {X -731.996,Y -2667.355,Z 1143.930,A -89.99946,B 0.00000,C 180.00000} ; outside
  LIN {X -731.996,Y -2667.355,Z 190.712,A -89.99946,B 0.00000,C 180.00000} ; preinsert
  LIN {X -731.996,Y -2667.355,Z -59.288,A -89.99946,B 0.00000,C 180.00000} ; insert
  LIN {X -731.996,Y -2667.355,Z -59.288,A -89.99946,B 0.00000,C 180.00000} ; release
  LIN {X -731.996,Y -2667.355,Z 240.712,A -89.99946,B 0.00000,C 180.00000} ; retreat
  ; Step 1947, bar 626
  LIN {X -606.996,Y -2667.355,Z 1143.930,A -89.99946,B 0.00000,C 180.00000} ; outside
  LIN {X -606.996,Y -2667.355,Z 190.712,A -89.99946,B 0.00000,C 180.00000} ; preinsert
  LIN {X -606.996,Y -2667.355,Z -59.288,A -89.99946,B 0.00000,C 180.00000} ; insert
  LIN {X -606.996,Y -2667.355,Z -59.288,A -89.99946,B 0.00000,C 180.00000} ; release
  LIN {X -606.996,Y -2667.355,Z 240.712,A -89.99946,B 0.00000,C 180.00000} ; retreat
  ; Step 1948, bar 624
  LIN {X -481.996,Y -2667.355,Z 1143.930,A -89.99946,B 0.00000,C 180.00000} ; outside
  LIN {X -481.996,Y -2667.355,Z 190.712,A -89.99946,B 0.00000,C 180.00000} ; preinsert
  LIN {X -481.996,Y -2667.355,Z -59.288,A -89.99946,B 0.00000,C 180.00000} ; insert
  LIN {X -481.996,Y -2667.355,Z -59.288,A -89.99946,B 0.00000,C 180.00000} ; release
  LIN {X -481.996,Y -2667.355,Z 240.712,A -89.99946,B 0.00000,C 180.00000} ; retreat
  ; Step 1949, bar 622
  LIN {X -356.996,Y -2667.355,Z 1143.930,A -89.99946,B 0.00000,C 180.00000} ; outside
  LIN {X -356.996,Y -2667.355,Z 190.712,A -89.99946,B 0.00000,C 180.00000} ; preinsert
  LIN {X -356.996,Y -2667.355,Z -59.288,A -89.99946,B 0.00000,C 180.00000} ; insert
  LIN {X -356.996,Y -2667.355,Z -59.288,A -89.99946,B 0.00000,C 180.00000} ; release
  LIN {X -356.996,Y -2667.355,Z 240.712,A -89.99946,B 0.00000,C 180.00000} ; retreat
  ; Step 1950, bar 620
  LIN {X -231.996,Y -2667.355,Z 1143.930,A -89.99946,B 0.00000,C 180.00000} ; outside
  LIN {X -231.996,Y -2667.355,Z 190.712,A -89.99946,B 0.00000,C 180.00000} ; preinsert
  LIN {X -231.996,Y -2667.355,Z -59.288,A -89.99946,B 0.00000,C 180.00000} ; insert
  LIN {X -231.996,Y -2667.355,Z -59.288,A -89.99946,B 0.00000,C 180.00000} ; release
  LIN {X -231.996,Y -2667.355,Z 240.712,A -89.99946,B 0.00000,C 180.00000} ; retreat
  ; Step 1951, bar 618
  LIN {X -106.996,Y -2667.355,Z 1143.930,A -89.99946,B 0.00000,C 180.00000} ; outside
  LIN {X -106.996,Y -2667.355,Z 190.712,A -89.99946,B 0.00000,C 180.00000} ; preinsert
  LIN {X -106.996,Y -2667.355,Z -59.288,A -89.99946,B 0.00000,C 180.00000} ; insert
  LIN {X -106.996,Y -2667.355,Z -59.288,A -89.99946,B 0.00000,C 180.00000} ; release
  LIN {X -106.996,Y -2667.355,Z 240.712,A -89.99946,B 0.00000,C 180.00000} ; retreat
  ; Step 1952, bar 597
  LIN {X -18.004,Y 2667.355,Z 1143.930,A 90.00054,B 0.00000,C 180.00000} ; outside
  LIN {X -18.004,Y 2667.355,Z 190.712,A 90.00054,B 0.00000,C 180.00000} ; preinsert
  LIN {X -18.004,Y 2667.355,Z -59.288,A 90.00054,B 0.00000,C 180.00000} ; insert
  LIN {X -18.004,Y 2667.355,Z -59.288,A 90.00054,B 0.00000,C 180.00000} ; release
  LIN {X -18.004,Y 2667.355,Z 240.712,A 90.00054,B 0.00000,C 180.00000} ; retreat
  ; Step 1953, bar 305
  LIN {X 106.996,Y 2667.355,Z 1143.930,A 90.00054,B 0.00000,C 180.00000} ; outside
  LIN {X 106.996,Y 2667.355,Z 190.712,A 90.00054,B 0.00000,C 180.00000} ; preinsert
  LIN {X 106.996,Y 2667.355,Z -59.288,A 90.00054,B 0.00000,C 180.00000} ; insert
  LIN {X 106.996,Y 2667.355,Z -59.288,A 90.00054,B 0.00000,C 180.00000} ; release
  LIN {X 106.996,Y 2667.355,Z 240.712,A 90.00054,B 0.00000,C 180.00000} ; retreat
  ; Step 1954, bar 333
  LIN {X 231.996,Y 2667.355,Z 1143.930,A 90.00054,B 0.00000,C 180.00000} ; outside
  LIN {X 231.996,Y 2667.355,Z 190.712,A 90.00054,B 0.00000,C 180.00000} ; preinsert
  LIN {X 231.996,Y 2667.355,Z -59.288,A 90.00054,B 0.00000,C 180.00000} ; insert
  LIN {X 231.996,Y 2667.355,Z -59.288,A 90.00054,B 0.00000,C 180.00000} ; release
  LIN {X 231.996,Y 2667.355,Z 240.712,A 90.00054,B 0.00000,C 180.00000} ; retreat
  ; Step 1955, bar 335
  LIN {X 356.996,Y 2667.355,Z 1143.930,A 90.00054,B 0.00000,C 180.00000} ; outside
  LIN {X 356.996,Y 2667.355,Z 190.712,A 90.00054,B 0.00000,C 180.00000} ; preinsert
  LIN {X 356.996,Y 2667.355,Z -59.288,A 90.00054,B 0.00000,C 180.00000} ; insert
  LIN {X 356.996,Y 2667.355,Z -59.288,A 90.00054,B 0.00000,C 180.00000} ; release
  LIN {X 356.996,Y 2667.355,Z 240.712,A 90.00054,B 0.00000,C 180.00000} ; retreat
  ; Step 1956, bar 337
  LIN {X 481.996,Y 2667.355,Z 1143.930,A 90.00054,B 0.00000,C 180.00000} ; outside
  LIN {X 481.996,Y 2667.355,Z 190.712,A 90.00054,B 0.00000,C 180.00000} ; preinsert
  LIN {X 481.996,Y 2667.355,Z -59.288,A 90.00054,B 0.00000,C 180.00000} ; insert
  LIN {X 481.996,Y 2667.355,Z -59.288,A 90.00054,B 0.00000,C 180.00000} ; release
  LIN {X 481.996,Y 2667.355,Z 240.712,A 90.00054,B 0.00000,C 180.00000} ; retreat
  ; Step 1957, bar 339
  LIN {X 606.996,Y 2667.355,Z 1143.930,A 90.00054,B 0.00000,C 180.00000} ; outside
  LIN {X 606.996,Y 2667.355,Z 190.712,A 90.00054,B 0.00000,C 180.00000} ; preinsert
  LIN {X 606.996,Y 2667.355,Z -59.288,A 90.00054,B 0.00000,C 180.00000} ; insert
  LIN {X 606.996,Y 2667.355,Z -59.288,A 90.00054,B 0.00000,C 180.00000} ; release
  LIN {X 606.996,Y 2667.355,Z 240.712,A 90.00054,B 0.00000,C 180.00000} ; retreat
  ; Step 1958, bar 341
  LIN {X 731.996,Y 2667.355,Z 1143.930,A 90.00054,B 0.00000,C 180.00000} ; outside
  LIN {X 731.996,Y 2667.355,Z 190.712,A 90.00054,B 0.00000,C 180.00000} ; preinsert
  LIN {X 731.996,Y 2667.355,Z -59.288,A 90.00054,B 0.00000,C 180.00000} ; insert
  LIN {X 731.996,Y 2667.355,Z -59.288,A 90.00054,B 0.00000,C 180.00000} ; release
  LIN {X 731.996,Y 2667.355,Z 240.712,A 90.00054,B 0.00000,C 180.00000} ; retreat
  ; Step 1959, bar 343
  LIN {X 856.996,Y 2667.355,Z 1143.930,A 90.00054,B 0.00000,C 180.00000} ; outside
  LIN {X 856.996,Y 2667.355,Z 190.712,A 90.00054,B 0.00000,C 180.00000} ; preinsert
  LIN {X 856.996,Y 2667.355,Z -59.288,A 90.00054,B 0.00000,C 180.00000} ; insert
  LIN {X 856.996,Y 2667.355,Z -59.288,A 90.00054,B 0.00000,C 180.00000} ; release
  LIN {X 856.996,Y 2667.355,Z 240.712,A 90.00054,B 0.00000,C 180.00000} ; retreat
  ; Step 1960, bar 345
  LIN {X 981.996,Y 2667.355,Z 1143.930,A 90.00054,B 0.00000,C 180.00000} ; outside
  LIN {X 981.996,Y 2667.355,Z 190.712,A 90.00054,B 0.00000,C 180.00000} ; preinsert
  LIN {X 981.996,Y 2667.355,Z -59.288,A 90.00054,B 0.00000,C 180.00000} ; insert
  LIN {X 981.996,Y 2667.355,Z -59.288,A 90.00054,B 0.00000,C 180.00000} ; release
  LIN {X 981.996,Y 2667.355,Z 240.712,A 90.00054,B 0.00000,C 180.00000} ; retreat
  ; Step 1961, bar 347
  LIN {X 1106.996,Y 2667.355,Z 1143.930,A 90.00054,B 0.00000,C 180.00000} ; outside
  LIN {X 1106.996,Y 2667.355,Z 190.712,A 90.00054,B 0.00000,C 180.00000} ; preinsert
  LIN {X 1106.996,Y 2667.355,Z -59.288,A 90.00054,B 0.00000,C 180.00000} ; insert
  LIN {X 1106.996,Y 2667.355,Z -59.288,A 90.00054,B 0.00000,C 180.00000} ; release
  LIN {X 1106.996,Y 2667.355,Z 240.712,A 90.00054,B 0.00000,C 180.00000} ; retreat
  ; Step 1962, bar 349
  LIN {X 1231.996,Y 2667.355,Z 1143.930,A 90.00054,B 0.00000,C 180.00000} ; outside
  LIN {X 1231.996,Y 2667.355,Z 190.712,A 90.00054,B 0.00000,C 180.00000} ; preinsert
  LIN {X 1231.996,Y 2667.355,Z -59.288,A 90.00054,B 0.00000,C 180.00000} ; insert
  LIN {X 1231.996,Y 2667.355,Z -59.288,A 90.00054,B 0.00000,C 180.00000} ; release
  LIN {X 1231.996,Y 2667.355,Z 240.712,A 90.00054,B 0.00000,C 180.00000} ; retreat
  ; Step 1963, bar 351
  LIN {X 1356.996,Y 2667.355,Z 1143.930,A 90.00054,B 0.00000,C 180.00000} ; outside
  LIN {X 1356.996,Y 2667.355,Z 190.712,A 90.00054,B 0.00000,C 180.00000} ; preinsert
  LIN {X 1356.996,Y 2667.355,Z -59.288,A 90.00054,B 0.00000,C 180.00000} ; insert
  LIN {X 1356.996,Y 2667.355,Z -59.288,A 90.00054,B 0.00000,C 180.00000} ; release
  LIN {X 1356.996,Y 2667.355,Z 240.712,A 90.00054,B 0.00000,C 180.00000} ; retreat
  ; Step 1964, bar 353
  LIN {X 1481.996,Y 2667.355,Z 1143.930,A 90.00054,B 0.00000,C 180.00000} ; outside
  LIN {X 1481.996,Y 2667.355,Z 190.712,A 90.00054,B 0.00000,C 180.00000} ; preinsert
  LIN {X 1481.996,Y 2667.355,Z -59.288,A 90.00054,B 0.00000,C 180.00000} ; insert
  LIN {X 1481.996,Y 2667.355,Z -59.288,A 90.00054,B 0.00000,C 180.00000} ; release
  LIN {X 1481.996,Y 2667.355,Z 240.712,A 90.00054,B 0.00000,C 180.00000} ; retreat
  ; Step 1965, bar 355
  LIN {X 1606.996,Y 2667.355,Z 1143.930,A 90.00054,B 0.00000,C 180.00000} ; outside
  LIN {X 1606.996,Y 2667.355,Z 190.712,A 90.00054,B 0.00000,C 180.00000} ; preinsert
  LIN {X 1606.996,Y 2667.355,Z -59.288,A 90.00054,B 0.00000,C 180.00000} ; insert
  LIN {X 1606.996,Y 2667.355,Z -59.288,A 90.00054,B 0.00000,C 180.00000} ; release
  LIN {X 1606.996,Y 2667.355,Z 240.712,A 90.00054,B 0.00000,C 180.00000} ; retreat
  ; Step 1966, bar 357
  LIN {X 1731.996,Y 2667.355,Z 1143.930,A 90.00054,B 0.00000,C 180.00000} ; outside
  LIN {X 1731.996,Y 2667.355,Z 190.712,A 90.00054,B 0.00000,C 180.00000} ; preinsert
  LIN {X 1731.996,Y 2667.355,Z -59.288,A 90.00054,B 0.00000,C 180.00000} ; insert
  LIN {X 1731.996,Y 2667.355,Z -59.288,A 90.00054,B 0.00000,C 180.00000} ; release
  LIN {X 1731.996,Y 2667.355,Z 240.712,A 90.00054,B 0.00000,C 180.00000} ; retreat
  ; Step 1967, bar 359
  LIN {X 1856.996,Y 2667.355,Z 1143.930,A 90.00054,B 0.00000,C 180.00000} ; outside
  LIN {X 1856.996,Y 2667.355,Z 190.712,A 90.00054,B 0.00000,C 180.00000} ; preinsert
  LIN {X 1856.996,Y 2667.355,Z -59.288,A 90.00054,B 0.00000,C 180.00000} ; insert
  LIN {X 1856.996,Y 2667.355,Z -59.288,A 90.00054,B 0.00000,C 180.00000} ; release
  LIN {X 1856.996,Y 2667.355,Z 240.712,A 90.00054,B 0.00000,C 180.00000} ; retreat
  ; Step 1968, bar 361
  LIN {X 2106.996,Y 2667.355,Z 1143.930,A 90.00054,B 0.00000,C 180.00000} ; outside
  LIN {X 2106.996,Y 2667.355,Z 190.712,A 90.00054,B 0.00000,C 180.00000} ; preinsert
  LIN {X 2106.996,Y 2667.355,Z -59.288,A 90.00054,B 0.00000,C 180.00000} ; insert
  LIN {X 2106.996,Y 2667.355,Z -59.288,A 90.00054,B 0.00000,C 180.00000} ; release
  LIN {X 2106.996,Y 2667.355,Z 240.712,A 90.00054,B 0.00000,C 180.00000} ; retreat
  ; Step 1969, bar 363
  LIN {X 2231.996,Y 2667.355,Z 1143.930,A 90.00054,B 0.00000,C 180.00000} ; outside
  LIN {X 2231.996,Y 2667.355,Z 190.712,A 90.00054,B 0.00000,C 180.00000} ; preinsert
  LIN {X 2231.996,Y 2667.355,Z -59.288,A 90.00054,B 0.00000,C 180.00000} ; insert
  LIN {X 2231.996,Y 2667.355,Z -59.288,A 90.00054,B 0.00000,C 180.00000} ; release
  LIN {X 2231.996,Y 2667.355,Z 240.712,A 90.00054,B 0.00000,C 180.00000} ; retreat
  ; Step 1970, bar 365
  LIN {X 2356.996,Y 2667.355,Z 1143.930,A 90.00054,B 0.00000,C 180.00000} ; outside
  LIN {X 2356.996,Y 2667.355,Z 190.712,A 90.00054,B 0.00000,C 180.00000} ; preinsert
  LIN {X 2356.996,Y 2667.355,Z -59.288,A 90.00054,B 0.00000,C 180.00000} ; insert
  LIN {X 2356.996,Y 2667.355,Z -59.288,A 90.00054,B 0.00000,C 180.00000} ; release
  LIN {X 2356.996,Y 2667.355,Z 240.712,A 90.00054,B 0.00000,C 180.00000} ; retreat
  ; Step 1971, bar 367
  LIN {X 2481.996,Y 2667.355,Z 1143.930,A 90.00054,B 0.00000,C 180.00000} ; outside
  LIN {X 2481.996,Y 2667.355,Z 190.712,A 90.00054,B 0.00000,C 180.00000} ; preinsert
  LIN {X 2481.996,Y 2667.355,Z -59.288,A 90.00054,B 0.00000,C 180.00000} ; insert
  LIN {X 2481.996,Y 2667.355,Z -59.288,A 90.00054,B 0.00000,C 180.00000} ; release
  LIN {X 2481.996,Y 2667.355,Z 240.712,A 90.00054,B 0.00000,C 180.00000} ; retreat
  ; Step 1972, bar 369
  LIN {X 2606.996,Y 2667.355,Z 1143.930,A 90.00054,B 0.00000,C 180.00000} ; outside
  LIN {X 2606.996,Y 2667.355,Z 190.712,A 90.00054,B 0.00000,C 180.00000} ; preinsert
  LIN {X 2606.996,Y 2667.355,Z -59.288,A 90.00054,B 0.00000,C 180.00000} ; insert
  LIN {X 2606.996,Y 2667.355,Z -59.288,A 90.00054,B 0.00000,C 180.00000} ; release
  LIN {X 2606.996,Y 2667.355,Z 240.712,A 90.00054,B 0.00000,C 180.00000} ; retreat
  ; Step 1973, bar 371
  LIN {X 2731.996,Y 2667.355,Z 1143.930,A 90.00054,B 0.00000,C 180.00000} ; outside
  LIN {X 2731.996,Y 2667.355,Z 190.712,A 90.00054,B 0.00000,C 180.00000} ; preinsert
  LIN {X 2731.996,Y 2667.355,Z -59.288,A 90.00054,B 0.00000,C 180.00000} ; insert
  LIN {X 2731.996,Y 2667.355,Z -59.288,A 90.00054,B 0.00000,C 180.00000} ; release
  LIN {X 2731.996,Y 2667.355,Z 240.712,A 90.00054,B 0.00000,C 180.00000} ; retreat
  ; Step 1974, bar 373
  LIN {X 2856.996,Y 2667.355,Z 1143.930,A 90.00054,B 0.00000,C 180.00000} ; outside
  LIN {X 2856.996,Y 2667.355,Z 190.712,A 90.00054,B 0.00000,C 180.00000} ; preinsert
  LIN {X 2856.996,Y 2667.355,Z -59.288,A 90.00054,B 0.00000,C 180.00000} ; insert
  LIN {X 2856.996,Y 2667.355,Z -59.288,A 90.00054,B 0.00000,C 180.00000} ; release
  LIN {X 2856.996,Y 2667.355,Z 240.712,A 90.00054,B 0.00000,C 180.00000} ; retreat
  ; Step 1975, bar 375
  LIN {X 2981.996,Y 2667.355,Z 1143.930,A 90.00054,B 0.00000,C 180.00000} ; outside
  LIN {X 2981.996,Y 2667.355,Z 190.712,A 90.00054,B 0.00000,C 180.00000} ; preinsert
  LIN {X 2981.996,Y 2667.355,Z -59.288,A 90.00054,B 0.00000,C 180.00000} ; insert
  LIN {X 2981.996,Y 2667.355,Z -59.288,A 90.00054,B 0.00000,C 180.00000} ; release
  LIN {X 2981.996,Y 2667.355,Z 240.712,A 90.00054,B 0.00000,C 180.00000} ; retreat
  ; Step 1976, bar 377
  LIN {X 3106.996,Y 2667.355,Z 1143.930,A 90.00054,B 0.00000,C 180.00000} ; outside
  LIN {X 3106.996,Y 2667.355,Z 190.712,A 90.00054,B 0.00000,C 180.00000} ; preinsert
  LIN {X 3106.996,Y 2667.355,Z -59.288,A 90.00054,B 0.00000,C 180.00000} ; insert
  LIN {X 3106.996,Y 2667.355,Z -59.288,A 90.00054,B 0.00000,C 180.00000} ; release
  LIN {X 3106.996,Y 2667.355,Z 240.712,A 90.00054,B 0.00000,C 180.00000} ; retreat
  ; Step 1977, bar 379
  LIN {X 3231.996,Y 2667.355,Z 1143.930,A 90.00054,B 0.00000,C 180.00000} ; outside
  LIN {X 3231.996,Y 2667.355,Z 190.712,A 90.00054,B 0.00000,C 180.00000} ; preinsert
  LIN {X 3231.996,Y 2667.355,Z -59.288,A 90.00054,B 0.00000,C 180.00000} ; insert
  LIN {X 3231.996,Y 2667.355,Z -59.288,A 90.00054,B 0.00000,C 180.00000} ; release
  LIN {X 3231.996,Y 2667.355,Z 240.712,A 90.00054,B 0.00000,C 180.00000} ; retreat
  ; Step 1978, bar 381
  LIN {X 3356.996,Y 2667.355,Z 1143.930,A 90.00054,B 0.00000,C 180.00000} ; outside
  LIN {X 3356.996,Y 2667.355,Z 190.712,A 90.00054,B 0.00000,C 180.00000} ; preinsert
  LIN {X 3356.996,Y 2667.355,Z -59.288,A 90.00054,B 0.00000,C 180.00000} ; insert
  LIN {X 3356.996,Y 2667.355,Z -59.288,A 90.00054,B 0.00000,C 180.00000} ; release
  LIN {X 3356.996,Y 2667.355,Z 240.712,A 90.00054,B 0.00000,C 180.00000} ; retreat
  ; Step 1979, bar 383
  LIN {X 3481.996,Y 2667.355,Z 1143.930,A 90.00054,B 0.00000,C 180.00000} ; outside
  LIN {X 3481.996,Y 2667.355,Z 190.712,A 90.00054,B 0.00000,C 180.00000} ; preinsert
  LIN {X 3481.996,Y 2667.355,Z -59.288,A 90.00054,B 0.00000,C 180.00000} ; insert
  LIN {X 3481.996,Y 2667.355,Z -59.288,A 90.00054,B 0.00000,C 180.00000} ; release
  LIN {X 3481.996,Y 2667.355,Z 240.712,A 90.00054,B 0.00000,C 180.00000} ; retreat
  ; Step 1980, bar 385
  LIN {X 3606.996,Y 2667.355,Z 1143.930,A 90.00054,B 0.00000,C 180.00000} ; outside
  LIN {X 3606.996,Y 2667.355,Z 190.712,A 90.00054,B 0.00000,C 180.00000} ; preinsert
  LIN {X 3606.996,Y 2667.355,Z -59.288,A 90.00054,B 0.00000,C 180.00000} ; insert
  LIN {X 3606.996,Y 2667.355,Z -59.288,A 90.00054,B 0.00000,C 180.00000} ; release
  LIN {X 3606.996,Y 2667.355,Z 240.712,A 90.00054,B 0.00000,C 180.00000} ; retreat
  ; Step 1981, bar 387
  LIN {X 3731.996,Y 2667.355,Z 1143.930,A 90.00054,B 0.00000,C 180.00000} ; outside
  LIN {X 3731.996,Y 2667.355,Z 190.712,A 90.00054,B 0.00000,C 180.00000} ; preinsert
  LIN {X 3731.996,Y 2667.355,Z -59.288,A 90.00054,B 0.00000,C 180.00000} ; insert
  LIN {X 3731.996,Y 2667.355,Z -59.288,A 90.00054,B 0.00000,C 180.00000} ; release
  LIN {X 3731.996,Y 2667.355,Z 240.712,A 90.00054,B 0.00000,C 180.00000} ; retreat
  ; Step 1982, bar 389
  LIN {X 3856.996,Y 2667.355,Z 1143.930,A 90.00054,B 0.00000,C 180.00000} ; outside
  LIN {X 3856.996,Y 2667.355,Z 190.712,A 90.00054,B 0.00000,C 180.00000} ; preinsert
  LIN {X 3856.996,Y 2667.355,Z -59.288,A 90.00054,B 0.00000,C 180.00000} ; insert
  LIN {X 3856.996,Y 2667.355,Z -59.288,A 90.00054,B 0.00000,C 180.00000} ; release
  LIN {X 3856.996,Y 2667.355,Z 240.712,A 90.00054,B 0.00000,C 180.00000} ; retreat
  ; Step 1983, bar 391
  LIN {X 3981.996,Y 2667.355,Z 1143.930,A 90.00054,B 0.00000,C 180.00000} ; outside
  LIN {X 3981.996,Y 2667.355,Z 190.712,A 90.00054,B 0.00000,C 180.00000} ; preinsert
  LIN {X 3981.996,Y 2667.355,Z -59.288,A 90.00054,B 0.00000,C 180.00000} ; insert
  LIN {X 3981.996,Y 2667.355,Z -59.288,A 90.00054,B 0.00000,C 180.00000} ; release
  LIN {X 3981.996,Y 2667.355,Z 240.712,A 90.00054,B 0.00000,C 180.00000} ; retreat
  ; Step 1984, bar 393
  LIN {X 4106.996,Y 2667.355,Z 1143.930,A 90.00054,B 0.00000,C 180.00000} ; outside
  LIN {X 4106.996,Y 2667.355,Z 190.712,A 90.00054,B 0.00000,C 180.00000} ; preinsert
  LIN {X 4106.996,Y 2667.355,Z -59.288,A 90.00054,B 0.00000,C 180.00000} ; insert
  LIN {X 4106.996,Y 2667.355,Z -59.288,A 90.00054,B 0.00000,C 180.00000} ; release
  LIN {X 4106.996,Y 2667.355,Z 240.712,A 90.00054,B 0.00000,C 180.00000} ; retreat
  ; Step 1985, bar 395
  LIN {X 4231.996,Y 2667.355,Z 1143.930,A 90.00054,B 0.00000,C 180.00000} ; outside
  LIN {X 4231.996,Y 2667.355,Z 190.712,A 90.00054,B 0.00000,C 180.00000} ; preinsert
  LIN {X 4231.996,Y 2667.355,Z -59.288,A 90.00054,B 0.00000,C 180.00000} ; insert
  LIN {X 4231.996,Y 2667.355,Z -59.288,A 90.00054,B 0.00000,C 180.00000} ; release
  LIN {X 4231.996,Y 2667.355,Z 240.712,A 90.00054,B 0.00000,C 180.00000} ; retreat
  ; Step 1986, bar 397
  LIN {X 4356.996,Y 2667.355,Z 1143.930,A 90.00054,B 0.00000,C 180.00000} ; outside
  LIN {X 4356.996,Y 2667.355,Z 190.712,A 90.00054,B 0.00000,C 180.00000} ; preinsert
  LIN {X 4356.996,Y 2667.355,Z -59.288,A 90.00054,B 0.00000,C 180.00000} ; insert
  LIN {X 4356.996,Y 2667.355,Z -59.288,A 90.00054,B 0.00000,C 180.00000} ; release
  LIN {X 4356.996,Y 2667.355,Z 240.712,A 90.00054,B 0.00000,C 180.00000} ; retreat
  ; Step 1987, bar 399
  LIN {X 4481.996,Y 2667.355,Z 1143.930,A 90.00054,B 0.00000,C 180.00000} ; outside
  LIN {X 4481.996,Y 2667.355,Z 190.712,A 90.00054,B 0.00000,C 180.00000} ; preinsert
  LIN {X 4481.996,Y 2667.355,Z -59.288,A 90.00054,B 0.00000,C 180.00000} ; insert
  LIN {X 4481.996,Y 2667.355,Z -59.288,A 90.00054,B 0.00000,C 180.00000} ; release
  LIN {X 4481.996,Y 2667.355,Z 240.712,A 90.00054,B 0.00000,C 180.00000} ; retreat
  ; Step 1988, bar 401
  LIN {X 4606.996,Y 2667.355,Z 1143.930,A 90.00054,B 0.00000,C 180.00000} ; outside
  LIN {X 4606.996,Y 2667.355,Z 190.712,A 90.00054,B 0.00000,C 180.00000} ; preinsert
  LIN {X 4606.996,Y 2667.355,Z -59.288,A 90.00054,B 0.00000,C 180.00000} ; insert
  LIN {X 4606.996,Y 2667.355,Z -59.288,A 90.00054,B 0.00000,C 180.00000} ; release
  LIN {X 4606.996,Y 2667.355,Z 240.712,A 90.00054,B 0.00000,C 180.00000} ; retreat
  ; Step 1989, bar 403
  LIN {X 4731.996,Y 2667.355,Z 1143.930,A 90.00054,B 0.00000,C 180.00000} ; outside
  LIN {X 4731.996,Y 2667.355,Z 190.712,A 90.00054,B 0.00000,C 180.00000} ; preinsert
  LIN {X 4731.996,Y 2667.355,Z -59.288,A 90.00054,B 0.00000,C 180.00000} ; insert
  LIN {X 4731.996,Y 2667.355,Z -59.288,A 90.00054,B 0.00000,C 180.00000} ; release
  LIN {X 4731.996,Y 2667.355,Z 240.712,A 90.00054,B 0.00000,C 180.00000} ; retreat
  ; Step 1990, bar 405
  LIN {X 4856.996,Y 2667.355,Z 1143.930,A 90.00054,B 0.00000,C 180.00000} ; outside
  LIN {X 4856.996,Y 2667.355,Z 190.712,A 90.00054,B 0.00000,C 180.00000} ; preinsert
  LIN {X 4856.996,Y 2667.355,Z -59.288,A 90.00054,B 0.00000,C 180.00000} ; insert
  LIN {X 4856.996,Y 2667.355,Z -59.288,A 90.00054,B 0.00000,C 180.00000} ; release
  LIN {X 4856.996,Y 2667.355,Z 240.712,A 90.00054,B 0.00000,C 180.00000} ; retreat
  ; Step 1991, bar 407
  LIN {X 4981.996,Y 2667.355,Z 1143.930,A 90.00054,B 0.00000,C 180.00000} ; outside
  LIN {X 4981.996,Y 2667.355,Z 190.712,A 90.00054,B 0.00000,C 180.00000} ; preinsert
  LIN {X 4981.996,Y 2667.355,Z -59.288,A 90.00054,B 0.00000,C 180.00000} ; insert
  LIN {X 4981.996,Y 2667.355,Z -59.288,A 90.00054,B 0.00000,C 180.00000} ; release
  LIN {X 4981.996,Y 2667.355,Z 240.712,A 90.00054,B 0.00000,C 180.00000} ; retreat
  ; Step 1992, bar 409
  LIN {X 5106.996,Y 2667.355,Z 1143.930,A 90.00054,B 0.00000,C 180.00000} ; outside
  LIN {X 5106.996,Y 2667.355,Z 190.712,A 90.00054,B 0.00000,C 180.00000} ; preinsert
  LIN {X 5106.996,Y 2667.355,Z -59.288,A 90.00054,B 0.00000,C 180.00000} ; insert
  LIN {X 5106.996,Y 2667.355,Z -59.288,A 90.00054,B 0.00000,C 180.00000} ; release
  LIN {X 5106.996,Y 2667.355,Z 240.712,A 90.00054,B 0.00000,C 180.00000} ; retreat
  ; Step 1993, bar 411
  LIN {X 5231.996,Y 2667.355,Z 1143.930,A 90.00054,B 0.00000,C 180.00000} ; outside
  LIN {X 5231.996,Y 2667.355,Z 190.712,A 90.00054,B 0.00000,C 180.00000} ; preinsert
  LIN {X 5231.996,Y 2667.355,Z -59.288,A 90.00054,B 0.00000,C 180.00000} ; insert
  LIN {X 5231.996,Y 2667.355,Z -59.288,A 90.00054,B 0.00000,C 180.00000} ; release
  LIN {X 5231.996,Y 2667.355,Z 240.712,A 90.00054,B 0.00000,C 180.00000} ; retreat
  ; Step 1994, bar 413
  LIN {X 5356.996,Y 2667.355,Z 1143.930,A 90.00054,B 0.00000,C 180.00000} ; outside
  LIN {X 5356.996,Y 2667.355,Z 190.712,A 90.00054,B 0.00000,C 180.00000} ; preinsert
  LIN {X 5356.996,Y 2667.355,Z -59.288,A 90.00054,B 0.00000,C 180.00000} ; insert
  LIN {X 5356.996,Y 2667.355,Z -59.288,A 90.00054,B 0.00000,C 180.00000} ; release
  LIN {X 5356.996,Y 2667.355,Z 240.712,A 90.00054,B 0.00000,C 180.00000} ; retreat
  ; Step 1995, bar 415
  LIN {X 5481.996,Y 2667.355,Z 1143.930,A 90.00054,B 0.00000,C 180.00000} ; outside
  LIN {X 5481.996,Y 2667.355,Z 190.712,A 90.00054,B 0.00000,C 180.00000} ; preinsert
  LIN {X 5481.996,Y 2667.355,Z -59.288,A 90.00054,B 0.00000,C 180.00000} ; insert
  LIN {X 5481.996,Y 2667.355,Z -59.288,A 90.00054,B 0.00000,C 180.00000} ; release
  LIN {X 5481.996,Y 2667.355,Z 240.712,A 90.00054,B 0.00000,C 180.00000} ; retreat
  ; Step 1996, bar 417
  LIN {X 5606.996,Y 2667.355,Z 1143.930,A 90.00054,B 0.00000,C 180.00000} ; outside
  LIN {X 5606.996,Y 2667.355,Z 190.712,A 90.00054,B 0.00000,C 180.00000} ; preinsert
  LIN {X 5606.996,Y 2667.355,Z -59.288,A 90.00054,B 0.00000,C 180.00000} ; insert
  LIN {X 5606.996,Y 2667.355,Z -59.288,A 90.00054,B 0.00000,C 180.00000} ; release
  LIN {X 5606.996,Y 2667.355,Z 240.712,A 90.00054,B 0.00000,C 180.00000} ; retreat
  ; Step 1997, bar 419
  LIN {X 5731.996,Y 2667.355,Z 1143.930,A 90.00054,B 0.00000,C 180.00000} ; outside
  LIN {X 5731.996,Y 2667.355,Z 190.712,A 90.00054,B 0.00000,C 180.00000} ; preinsert
  LIN {X 5731.996,Y 2667.355,Z -59.288,A 90.00054,B 0.00000,C 180.00000} ; insert
  LIN {X 5731.996,Y 2667.355,Z -59.288,A 90.00054,B 0.00000,C 180.00000} ; release
  LIN {X 5731.996,Y 2667.355,Z 240.712,A 90.00054,B 0.00000,C 180.00000} ; retreat
  ; Step 1998, bar 421
  LIN {X 5856.996,Y 2667.355,Z 1143.930,A 90.00054,B 0.00000,C 180.00000} ; outside
  LIN {X 5856.996,Y 2667.355,Z 190.712,A 90.00054,B 0.00000,C 180.00000} ; preinsert
  LIN {X 5856.996,Y 2667.355,Z -59.288,A 90.00054,B 0.00000,C 180.00000} ; insert
  LIN {X 5856.996,Y 2667.355,Z -59.288,A 90.00054,B 0.00000,C 180.00000} ; release
  LIN {X 5856.996,Y 2667.355,Z 240.712,A 90.00054,B 0.00000,C 180.00000} ; retreat
  ; Step 1999, bar 423
  LIN {X 6106.996,Y 2667.355,Z 1143.930,A 90.00054,B 0.00000,C 180.00000} ; outside
  LIN {X 6106.996,Y 2667.355,Z 190.712,A 90.00054,B 0.00000,C 180.00000} ; preinsert
  LIN {X 6106.996,Y 2667.355,Z -59.288,A 90.00054,B 0.00000,C 180.00000} ; insert
  LIN {X 6106.996,Y 2667.355,Z -59.288,A 90.00054,B 0.00000,C 180.00000} ; release
  LIN {X 6106.996,Y 2667.355,Z 240.712,A 90.00054,B 0.00000,C 180.00000} ; retreat
  ; Step 2000, bar 425
  LIN {X 6231.996,Y 2667.355,Z 1143.930,A 90.00054,B 0.00000,C 180.00000} ; outside
  LIN {X 6231.996,Y 2667.355,Z 190.712,A 90.00054,B 0.00000,C 180.00000} ; preinsert
  LIN {X 6231.996,Y 2667.355,Z -59.288,A 90.00054,B 0.00000,C 180.00000} ; insert
  LIN {X 6231.996,Y 2667.355,Z -59.288,A 90.00054,B 0.00000,C 180.00000} ; release
  LIN {X 6231.996,Y 2667.355,Z 240.712,A 90.00054,B 0.00000,C 180.00000} ; retreat
  ; Step 2001, bar 427
  LIN {X 6356.996,Y 2667.355,Z 1143.930,A 90.00054,B 0.00000,C 180.00000} ; outside
  LIN {X 6356.996,Y 2667.355,Z 190.712,A 90.00054,B 0.00000,C 180.00000} ; preinsert
  LIN {X 6356.996,Y 2667.355,Z -59.288,A 90.00054,B 0.00000,C 180.00000} ; insert
  LIN {X 6356.996,Y 2667.355,Z -59.288,A 90.00054,B 0.00000,C 180.00000} ; release
  LIN {X 6356.996,Y 2667.355,Z 240.712,A 90.00054,B 0.00000,C 180.00000} ; retreat
  ; Step 2002, bar 429
  LIN {X 6481.996,Y 2667.355,Z 1143.930,A 90.00054,B 0.00000,C 180.00000} ; outside
  LIN {X 6481.996,Y 2667.355,Z 190.712,A 90.00054,B 0.00000,C 180.00000} ; preinsert
  LIN {X 6481.996,Y 2667.355,Z -59.288,A 90.00054,B 0.00000,C 180.00000} ; insert
  LIN {X 6481.996,Y 2667.355,Z -59.288,A 90.00054,B 0.00000,C 180.00000} ; release
  LIN {X 6481.996,Y 2667.355,Z 240.712,A 90.00054,B 0.00000,C 180.00000} ; retreat
  ; Step 2003, bar 431
  LIN {X 6606.996,Y 2667.355,Z 1143.930,A 90.00054,B 0.00000,C 180.00000} ; outside
  LIN {X 6606.996,Y 2667.355,Z 190.712,A 90.00054,B 0.00000,C 180.00000} ; preinsert
  LIN {X 6606.996,Y 2667.355,Z -59.288,A 90.00054,B 0.00000,C 180.00000} ; insert
  LIN {X 6606.996,Y 2667.355,Z -59.288,A 90.00054,B 0.00000,C 180.00000} ; release
  LIN {X 6606.996,Y 2667.355,Z 240.712,A 90.00054,B 0.00000,C 180.00000} ; retreat
  ; Step 2004, bar 433
  LIN {X 6731.996,Y 2667.355,Z 1143.930,A 90.00054,B 0.00000,C 180.00000} ; outside
  LIN {X 6731.996,Y 2667.355,Z 190.712,A 90.00054,B 0.00000,C 180.00000} ; preinsert
  LIN {X 6731.996,Y 2667.355,Z -59.288,A 90.00054,B 0.00000,C 180.00000} ; insert
  LIN {X 6731.996,Y 2667.355,Z -59.288,A 90.00054,B 0.00000,C 180.00000} ; release
  LIN {X 6731.996,Y 2667.355,Z 240.712,A 90.00054,B 0.00000,C 180.00000} ; retreat
  ; Step 2005, bar 435
  LIN {X 6856.996,Y 2667.355,Z 1143.930,A 90.00054,B 0.00000,C 180.00000} ; outside
  LIN {X 6856.996,Y 2667.355,Z 190.712,A 90.00054,B 0.00000,C 180.00000} ; preinsert
  LIN {X 6856.996,Y 2667.355,Z -59.288,A 90.00054,B 0.00000,C 180.00000} ; insert
  LIN {X 6856.996,Y 2667.355,Z -59.288,A 90.00054,B 0.00000,C 180.00000} ; release
  LIN {X 6856.996,Y 2667.355,Z 240.712,A 90.00054,B 0.00000,C 180.00000} ; retreat
  ; Step 2006, bar 437
  LIN {X 6981.996,Y 2667.355,Z 1143.930,A 90.00054,B 0.00000,C 180.00000} ; outside
  LIN {X 6981.996,Y 2667.355,Z 190.712,A 90.00054,B 0.00000,C 180.00000} ; preinsert
  LIN {X 6981.996,Y 2667.355,Z -59.288,A 90.00054,B 0.00000,C 180.00000} ; insert
  LIN {X 6981.996,Y 2667.355,Z -59.288,A 90.00054,B 0.00000,C 180.00000} ; release
  LIN {X 6981.996,Y 2667.355,Z 240.712,A 90.00054,B 0.00000,C 180.00000} ; retreat
  ; Step 2007, bar 439
  LIN {X 7106.996,Y 2667.355,Z 1143.930,A 90.00054,B 0.00000,C 180.00000} ; outside
  LIN {X 7106.996,Y 2667.355,Z 190.712,A 90.00054,B 0.00000,C 180.00000} ; preinsert
  LIN {X 7106.996,Y 2667.355,Z -59.288,A 90.00054,B 0.00000,C 180.00000} ; insert
  LIN {X 7106.996,Y 2667.355,Z -59.288,A 90.00054,B 0.00000,C 180.00000} ; release
  LIN {X 7106.996,Y 2667.355,Z 240.712,A 90.00054,B 0.00000,C 180.00000} ; retreat
  ; Step 2008, bar 441
  LIN {X 7231.996,Y 2667.355,Z 1143.930,A 90.00054,B 0.00000,C 180.00000} ; outside
  LIN {X 7231.996,Y 2667.355,Z 190.712,A 90.00054,B 0.00000,C 180.00000} ; preinsert
  LIN {X 7231.996,Y 2667.355,Z -59.288,A 90.00054,B 0.00000,C 180.00000} ; insert
  LIN {X 7231.996,Y 2667.355,Z -59.288,A 90.00054,B 0.00000,C 180.00000} ; release
  LIN {X 7231.996,Y 2667.355,Z 240.712,A 90.00054,B 0.00000,C 180.00000} ; retreat
  ; Step 2009, bar 443
  LIN {X 7356.996,Y 2667.355,Z 1143.930,A 90.00054,B 0.00000,C 180.00000} ; outside
  LIN {X 7356.996,Y 2667.355,Z 190.712,A 90.00054,B 0.00000,C 180.00000} ; preinsert
  LIN {X 7356.996,Y 2667.355,Z -59.288,A 90.00054,B 0.00000,C 180.00000} ; insert
  LIN {X 7356.996,Y 2667.355,Z -59.288,A 90.00054,B 0.00000,C 180.00000} ; release
  LIN {X 7356.996,Y 2667.355,Z 240.712,A 90.00054,B 0.00000,C 180.00000} ; retreat
  ; Step 2010, bar 445
  LIN {X 7481.996,Y 2667.355,Z 1143.930,A 90.00054,B 0.00000,C 180.00000} ; outside
  LIN {X 7481.996,Y 2667.355,Z 190.712,A 90.00054,B 0.00000,C 180.00000} ; preinsert
  LIN {X 7481.996,Y 2667.355,Z -59.288,A 90.00054,B 0.00000,C 180.00000} ; insert
  LIN {X 7481.996,Y 2667.355,Z -59.288,A 90.00054,B 0.00000,C 180.00000} ; release
  LIN {X 7481.996,Y 2667.355,Z 240.712,A 90.00054,B 0.00000,C 180.00000} ; retreat
  ; Step 2011, bar 447
  LIN {X 7606.996,Y 2667.355,Z 1143.930,A 90.00054,B 0.00000,C 180.00000} ; outside
  LIN {X 7606.996,Y 2667.355,Z 190.712,A 90.00054,B 0.00000,C 180.00000} ; preinsert
  LIN {X 7606.996,Y 2667.355,Z -59.288,A 90.00054,B 0.00000,C 180.00000} ; insert
  LIN {X 7606.996,Y 2667.355,Z -59.288,A 90.00054,B 0.00000,C 180.00000} ; release
  LIN {X 7606.996,Y 2667.355,Z 240.712,A 90.00054,B 0.00000,C 180.00000} ; retreat
  ; Step 2012, bar 449
  LIN {X 7731.996,Y 2667.355,Z 1143.930,A 90.00054,B 0.00000,C 180.00000} ; outside
  LIN {X 7731.996,Y 2667.355,Z 190.712,A 90.00054,B 0.00000,C 180.00000} ; preinsert
  LIN {X 7731.996,Y 2667.355,Z -59.288,A 90.00054,B 0.00000,C 180.00000} ; insert
  LIN {X 7731.996,Y 2667.355,Z -59.288,A 90.00054,B 0.00000,C 180.00000} ; release
  LIN {X 7731.996,Y 2667.355,Z 240.712,A 90.00054,B 0.00000,C 180.00000} ; retreat
  ; Step 2013, bar 451
  LIN {X 7856.996,Y 2667.355,Z 1143.930,A 90.00054,B 0.00000,C 180.00000} ; outside
  LIN {X 7856.996,Y 2667.355,Z 190.712,A 90.00054,B 0.00000,C 180.00000} ; preinsert
